ABB RobotStudio station: robotic-ABB-Cake-Simulation-Final.rspag

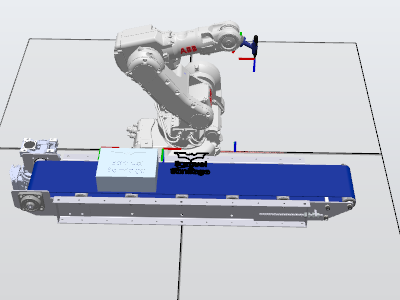
--- station ---
Station robotic-ABB-Cake (saved by RobotStudio 25.3.11371.0)
Controller IRB140_6_81
  mechanical unit ROB_1: IRB140_6_81_C_03, 6 joints, base frame (0, 0, 0) mm
Layout (positions relative to the parent item):
  - IRB140_6_81_C_03 [mechanism, from %ABB.RobotStudio.Models.IRB140%\IRB140_6_81_C_G_03.rslib] at (0, 0, 0) mm; joint values [0, -0.726, 0.4848, 0, 0.7648, 0] (rad or m)
  - Marker [mechanism] at (256.29, 0, 679.5) mm, rotated rx 180 ry 60 rz 180 deg
      TCP Marker at (50.06, 0, 105.48) mm, rotated rx 0 ry 60 rz 0 deg
      links: Marker-Tool
  - Box_Names [part] at (-315, -770, 485) mm, size 230 x 165 x 83 mm
  - Conveyor [part] at (358.05, -804.87, 88.69) mm, rotated rx 0 ry 0 rz 90 deg, size 367.7 x 1444.4 x 354.2 mm
  - SmartComponent_1 [smart component]
      signals: DI DI01, DI DI02, DI DI03, DI Conveyor_FWD, DI Conveyor_INV, DO DI_01, DO DI_02, DO DI_03
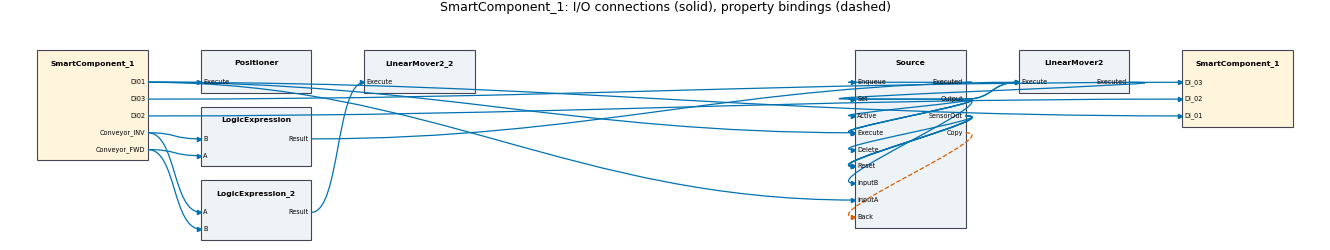
      connections:
        Source.Executed -> Queue.Enqueue
        LinearMover2.Executed -> LogicSRLatch.Set
        LogicSRLatch.Output -> Timer.Active
        Timer.Output -> LogicSRLatch_2.Set
        LogicSRLatch_2.Output -> LinearMover.Execute
        LineSensor.SensorOut -> Queue.Delete
        LineSensor.SensorOut -> Timer.Reset
        LineSensor.SensorOut -> LogicSRLatch.Reset
        LineSensor.SensorOut -> LogicSRLatch_2.Reset
        Repeater.Output -> LinearMover2.Execute
        Repeater.Output -> Source.Execute
        Timer_2.Output -> LogicGate.InputB
        LogicSRLatch_3.Output -> Source.Execute
        LogicSRLatch_3.Output -> LinearMover2.Execute
        LogicGate.Output -> LogicSRLatch_3.Set
        LineSensor.SensorOut -> LogicSRLatch_3.Reset
        SmartComponent_1.DI01 -> ?.Execute
        SmartComponent_1.DI01 -> LogicGate.InputA
        SmartComponent_1.DI03 -> SmartComponent_1.DI_03
        SmartComponent_1.DI02 -> SmartComponent_1.DI_02
        SmartComponent_1.DI01 -> SmartComponent_1.DI_01
        SmartComponent_1.Conveyor_INV -> LogicExpression.B
        SmartComponent_1.Conveyor_FWD -> LogicExpression.A
        LogicExpression.Result -> LinearMover2.Execute
        SmartComponent_1.Conveyor_INV -> LogicExpression_2.A
        SmartComponent_1.Conveyor_FWD -> LogicExpression_2.B
        LogicExpression_2.Result -> LinearMover2_2.Execute
        SmartComponent_1.DI01 -> Positioner.Execute
        Source.Copy => Queue.Back
    - LinearMover2 [smart component, from Components\LinearMover2.rslib]
        properties: Object=Box_Names; Direction=[1 0 0]; Distance=0.25; Duration=3; Reference=Global; ReferenceObject=(none)
    - LogicExpression [smart component, from Components\LogicExpression.rslib]
        properties: Expression=A AND NOT B
    - Positioner [smart component, from Components\Positioner.rslib]
        properties: Object=Box_Names; Position=[-0.315 -0.77 0.485]; Orientation=[0 0 0]; Reference=Global; ReferenceObject=(none)
    - LinearMover2_2 [smart component, from Components\LinearMover2.rslib]
        properties: Object=Box_Names; Direction=[-1 0 0]; Distance=0.5; Duration=8.5; Reference=Global; ReferenceObject=(none)
    - LogicExpression_2 [smart component, from Components\LogicExpression.rslib]
        properties: Expression=A AND NOT B
Attachment: Marker is attached to IRB140_6_81_C_03 / Link6
Attachment: Cake is attached to Box_Names
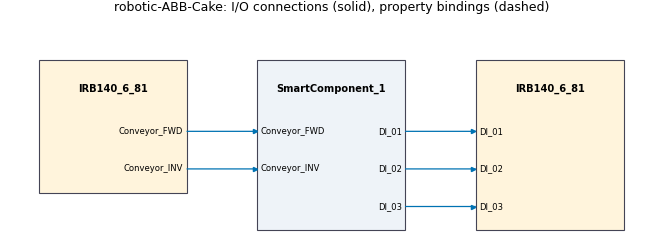
Station logic (signal -> signal, property => property):
  IRB140_6_81.Conveyor_FWD -> SmartComponent_1.Conveyor_FWD
  IRB140_6_81.Conveyor_INV -> SmartComponent_1.Conveyor_INV
  SmartComponent_1.DI_01 -> IRB140_6_81.DI_01
  SmartComponent_1.DI_02 -> IRB140_6_81.DI_02
  SmartComponent_1.DI_03 -> IRB140_6_81.DI_03

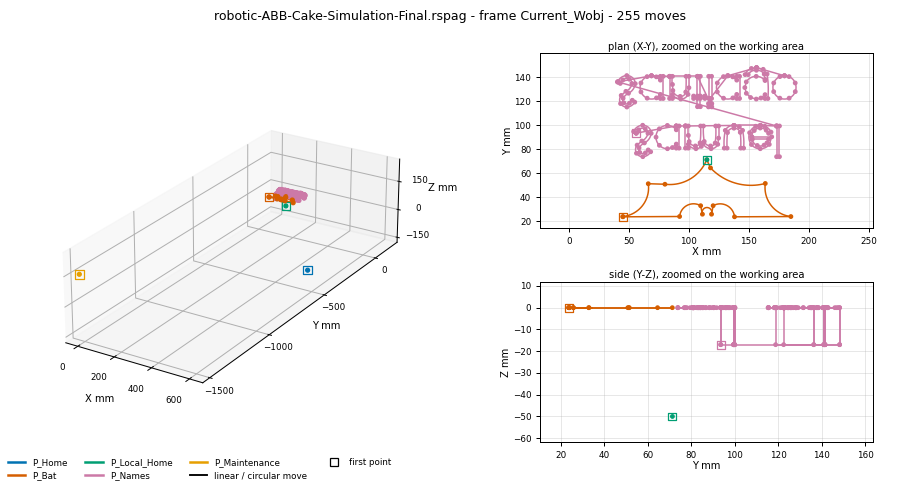
[picture p0: tool path of robotic-ABB-Cake-Simulation-Final.rspag in frame Current_Wobj, 255 of 255 moves have a stored position in this frame; points joined in program order, loops and branches not executed]
--- Controller Data/IRB140_6_81/RAPID/TASK1/PROGMOD/CalibData.mod ---
MODULE CalibData
ENDMODULE

--- Controller Data/IRB140_6_81/RAPID/TASK1/PROGMOD/Module1.mod ---
MODULE Module1
    !DATA
    !Homes
    CONST robtarget T_Home:=[[637.610974939,-605,-15.40043816],[0,0,0,1],[0,0,0,0],[9E+09,9E+09,9E+09,9E+09,9E+09,9E+09]];
    CONST robtarget T_Local_Home:=[[115.079,71.263,-50],[0.707106781,0.000000005,-0.000000005,-0.707106781],[0,0,0,0],[9E+09,9E+09,9E+09,9E+09,9E+09,9E+09]];

    !Batman Icon
    CONST robtarget Target_290:=[[44.887375283,23.575,0],[0.707106781,0,0,-0.707106781],[0,0,0,0],[9E+09,9E+09,9E+09,9E+09,9E+09,9E+09]];
    CONST robtarget Target_300:=[[92.217626762,23.834877014,0],[0.5,0,0,-0.866025404],[-1,0,-1,0],[9E+09,9E+09,9E+09,9E+09,9E+09,9E+09]];
    CONST robtarget Target_400:=[[168.340891695,33.478608179,0],[0.5,0,0,-0.866025404],[-1,0,-1,0],[9E+09,9E+09,9E+09,9E+09,9E+09,9E+09]];
    CONST robtarget Target_430:=[[118.021503486,64.425747652,0],[0.5,0,0,-0.866025404],[0,0,0,0],[9E+09,9E+09,9E+09,9E+09,9E+09,9E+09]];
    CONST robtarget Target_310:=[[97.860623741,32.777873993,0],[0.5,0,0,-0.866025404],[-1,0,-1,0],[9E+09,9E+09,9E+09,9E+09,9E+09,9E+09]];
    CONST robtarget Target_480:=[[61.659109682,33.478608179,0],[0.5,0,0,-0.866025404],[-1,0,-1,0],[9E+09,9E+09,9E+09,9E+09,9E+09,9E+09]];
    CONST robtarget Target_420:=[[135.262514114,52.897562122,0],[0.5,0,0,-0.866025404],[-1,0,-1,0],[9E+09,9E+09,9E+09,9E+09,9E+09,9E+09]];
    CONST robtarget Target_460:=[[79.985840188,50.770867258,0],[0.5,0,0,-0.866025404],[0,0,0,0],[9E+09,9E+09,9E+09,9E+09,9E+09,9E+09]];
    CONST robtarget Target_330:=[[111.283377266,25.744747734,0],[0.5,0,0,-0.866025404],[-1,0,-1,0],[9E+09,9E+09,9E+09,9E+09,9E+09,9E+09]];
    CONST robtarget Target_380:=[[138.079373741,23.575,0],[0.5,0,0,-0.866025404],[0,0,0,0],[9E+09,9E+09,9E+09,9E+09,9E+09,9E+09]];
    CONST robtarget Target_340:=[[112.525,30.426625252,0],[0.5,0,0,-0.866025404],[-1,0,-1,0],[9E+09,9E+09,9E+09,9E+09,9E+09,9E+09]];
    CONST robtarget Target_490:=[[44.854375315,23.789501762,0],[0.707106781,0,0,-0.707106781],[0,0,0,0],[9E+09,9E+09,9E+09,9E+09,9E+09,9E+09]];
    CONST robtarget Target_360:=[[120.205747986,32.852127266,0],[0.5,0,0,-0.866025404],[-1,0,-1,0],[9E+09,9E+09,9E+09,9E+09,9E+09,9E+09]];
    CONST robtarget Target_350:=[[118.898123741,25.740625,0],[0.5,0,0,-0.866025404],[0,0,0,0],[9E+09,9E+09,9E+09,9E+09,9E+09,9E+09]];
    CONST robtarget Target_370:=[[132.139376259,32.777873993,0],[0.5,0,0,-0.866025404],[-1,0,-1,0],[9E+09,9E+09,9E+09,9E+09,9E+09,9E+09]];
    CONST robtarget Target_410:=[[163.773995972,51.414627266,0],[0.5,0,0,-0.866025404],[0,0,0,0],[9E+09,9E+09,9E+09,9E+09,9E+09,9E+09]];
    CONST robtarget Target_470:=[[66.061000252,51.208377266,0],[0.5,0,0,-0.866025404],[-1,0,-1,0],[9E+09,9E+09,9E+09,9E+09,9E+09,9E+09]];
    CONST robtarget Target_320:=[[109.794252014,32.852127266,0],[0.5,0,0,-0.866025404],[0,0,0,0],[9E+09,9E+09,9E+09,9E+09,9E+09,9E+09]];
    CONST robtarget Target_440:=[[114.884500504,71.210504532,0],[0.5,0,0,-0.866025404],[-1,0,-1,0],[9E+09,9E+09,9E+09,9E+09,9E+09,9E+09]];
    CONST robtarget Target_450:=[[101.522546531,55.448907324,0],[0.5,0,0,-0.866025404],[-1,0,-1,0],[9E+09,9E+09,9E+09,9E+09,9E+09,9E+09]];
    CONST robtarget Target_390:=[[185.145619965,23.789501762,0],[0.5,0,0,-0.866025404],[-1,0,-1,0],[9E+09,9E+09,9E+09,9E+09,9E+09,9E+09]];

    !Nombres
    CONST robtarget Names_00:=[[55.976,93.47,-17],[0.707106781,0,0,-0.707106781],[0,0,0,0],[9E+09,9E+09,9E+09,9E+09,9E+09,9E+09]];
    CONST robtarget Names_10:=[[55.976,93.47,0],[0.707106781,0,0,-0.707106781],[-1,-1,0,0],[9E+09,9E+09,9E+09,9E+09,9E+09,9E+09]];
    CONST robtarget Names_20:=[[53.851,94.745,0],[0.707106781,0,0,-0.707106781],[-1,-1,0,0],[9E+09,9E+09,9E+09,9E+09,9E+09,9E+09]];
    CONST robtarget Names_30:=[[57.267,98.815,0],[0.707106781,0,0,-0.707106781],[-1,-1,0,0],[9E+09,9E+09,9E+09,9E+09,9E+09,9E+09]];
    CONST robtarget Names_40:=[[61.397,100.031,0],[0.707106781,0,0,-0.707106781],[-1,-1,0,0],[9E+09,9E+09,9E+09,9E+09,9E+09,9E+09]];
    CONST robtarget Names_50:=[[66.419,98.025,0],[0.707106781,0,0,-0.707106781],[-1,-1,0,0],[9E+09,9E+09,9E+09,9E+09,9E+09,9E+09]];
    CONST robtarget Names_60:=[[68.484,93.3,0],[0.707106781,0,0,-0.707106781],[-1,-1,0,0],[9E+09,9E+09,9E+09,9E+09,9E+09,9E+09]];
    CONST robtarget Names_70:=[[67.277,89.545,0],[0.707106781,0,0,-0.707106781],[-1,-1,0,0],[9E+09,9E+09,9E+09,9E+09,9E+09,9E+09]];
    CONST robtarget Names_80:=[[62.825,85.279,0],[0.707106781,0,0,-0.707106781],[-1,-1,0,0],[9E+09,9E+09,9E+09,9E+09,9E+09,9E+09]];
    CONST robtarget Names_90:=[[59.596,82.78,0],[0.707106781,0,0,-0.707106781],[-1,-1,0,0],[9E+09,9E+09,9E+09,9E+09,9E+09,9E+09]];
    CONST robtarget Names_100:=[[58.355,81.115,0],[0.707106781,0,0,-0.707106781],[-1,-1,0,0],[9E+09,9E+09,9E+09,9E+09,9E+09,9E+09]];
    CONST robtarget Names_110:=[[58.015,79.534,0],[0.707106781,0,0,-0.707106781],[-1,-1,0,0],[9E+09,9E+09,9E+09,9E+09,9E+09,9E+09]];
    CONST robtarget Names_120:=[[58.975,77.274,0],[0.707106781,0,0,-0.707106781],[-1,-1,0,0],[9E+09,9E+09,9E+09,9E+09,9E+09,9E+09]];
    CONST robtarget Names_130:=[[61.448,76.356,0],[0.707106781,0,0,-0.707106781],[-1,-1,0,0],[9E+09,9E+09,9E+09,9E+09,9E+09,9E+09]];
    CONST robtarget Names_140:=[[63.615,76.951,0],[0.707106781,0,0,-0.707106781],[-1,-1,0,0],[9E+09,9E+09,9E+09,9E+09,9E+09,9E+09]];
    CONST robtarget Names_150:=[[66.02,79.415,0],[0.707106781,0,0,-0.707106781],[-1,-1,0,0],[9E+09,9E+09,9E+09,9E+09,9E+09,9E+09]];
    CONST robtarget Names_160:=[[68.059,77.869,0],[0.707106781,0,0,-0.707106781],[-1,-1,0,0],[9E+09,9E+09,9E+09,9E+09,9E+09,9E+09]];
    CONST robtarget Names_170:=[[64.805,74.648,0],[0.707106781,0,0,-0.707106781],[-1,-1,0,0],[9E+09,9E+09,9E+09,9E+09,9E+09,9E+09]];
    CONST robtarget Names_180:=[[61.499,73.773,0],[0.707106781,0,0,-0.707106781],[-1,-1,0,0],[9E+09,9E+09,9E+09,9E+09,9E+09,9E+09]];
    CONST robtarget Names_190:=[[58.414,74.546,0],[0.707106781,0,0,-0.707106781],[-1,-1,0,0],[9E+09,9E+09,9E+09,9E+09,9E+09,9E+09]];
    CONST robtarget Names_200:=[[56.213,76.662,0],[0.707106781,0,0,-0.707106781],[-1,-1,0,0],[9E+09,9E+09,9E+09,9E+09,9E+09,9E+09]];
    CONST robtarget Names_210:=[[55.432,79.636,0],[0.707106781,0,0,-0.707106781],[-1,-1,0,0],[9E+09,9E+09,9E+09,9E+09,9E+09,9E+09]];
    CONST robtarget Names_220:=[[56.757,83.46,0],[0.707106781,0,0,-0.707106781],[-1,-1,0,0],[9E+09,9E+09,9E+09,9E+09,9E+09,9E+09]];
    CONST robtarget Names_230:=[[60.649,86.876,0],[0.707106781,0,0,-0.707106781],[-1,-1,0,0],[9E+09,9E+09,9E+09,9E+09,9E+09,9E+09]];
    CONST robtarget Names_240:=[[64.932,90.887,0],[0.707106781,0,0,-0.707106781],[-1,-1,0,0],[9E+09,9E+09,9E+09,9E+09,9E+09,9E+09]];
    CONST robtarget Names_250:=[[65.782,93.351,0],[0.707106781,0,0,-0.707106781],[-1,-1,0,0],[9E+09,9E+09,9E+09,9E+09,9E+09,9E+09]];
    CONST robtarget Names_260:=[[65.204,95.442,0],[0.707106781,0,0,-0.707106781],[-1,-1,0,0],[9E+09,9E+09,9E+09,9E+09,9E+09,9E+09]];
    CONST robtarget Names_270:=[[63.521,97.014,0],[0.707106781,0,0,-0.707106781],[-1,-1,0,0],[9E+09,9E+09,9E+09,9E+09,9E+09,9E+09]];
    CONST robtarget Names_280:=[[61.159,97.6,0],[0.707106781,0,0,-0.707106781],[-1,-1,0,0],[9E+09,9E+09,9E+09,9E+09,9E+09,9E+09]];
    CONST robtarget Names_290:=[[58.019,96.283,0],[0.707106781,0,0,-0.707106781],[-1,-1,0,0],[9E+09,9E+09,9E+09,9E+09,9E+09,9E+09]];
    CONST robtarget Names_300:=[[55.976,93.47,0],[0.707106781,0,0,-0.707106781],[-1,-1,0,0],[9E+09,9E+09,9E+09,9E+09,9E+09,9E+09]];
    CONST robtarget Names_310:=[[55.976,93.47,-17],[0.707106781,0,0,-0.707106781],[-1,-1,0,0],[9E+09,9E+09,9E+09,9E+09,9E+09,9E+09]];
    CONST robtarget Names_320:=[[89.456,99.402,-17],[0.608761429,0,0,-0.79335334],[-1,0,-1,0],[9E+09,9E+09,9E+09,9E+09,9E+09,9E+09]];
    CONST robtarget Names_330:=[[89.456,99.402,0],[0.608761429,0,0,-0.79335334],[-1,0,-1,0],[9E+09,9E+09,9E+09,9E+09,9E+09,9E+09]];
    CONST robtarget Names_340:=[[89.456,96.224,0],[0.608761429,0,0,-0.79335334],[-1,0,-1,0],[9E+09,9E+09,9E+09,9E+09,9E+09,9E+09]];
    CONST robtarget Names_350:=[[86.1,98.96,0],[0.608761429,0,0,-0.79335334],[-1,0,-1,0],[9E+09,9E+09,9E+09,9E+09,9E+09,9E+09]];
    CONST robtarget Names_360:=[[82.029,99.878,0],[0.608761429,0,0,-0.79335334],[-1,0,-1,0],[9E+09,9E+09,9E+09,9E+09,9E+09,9E+09]];
    CONST robtarget Names_370:=[[78.378,99.161,0],[0.608761429,0,0,-0.79335334],[-1,0,-1,0],[9E+09,9E+09,9E+09,9E+09,9E+09,9E+09]];
    CONST robtarget Names_380:=[[75.325,97.031,0],[0.608761429,0,0,-0.79335334],[-1,0,-1,0],[9E+09,9E+09,9E+09,9E+09,9E+09,9E+09]];
    CONST robtarget Names_390:=[[73.231,93.852,0],[0.608761429,0,0,-0.79335334],[-1,0,-1,0],[9E+09,9E+09,9E+09,9E+09,9E+09,9E+09]];
    CONST robtarget Names_400:=[[72.546,90.105,0],[0.608761429,0,0,-0.79335334],[-1,0,-1,0],[9E+09,9E+09,9E+09,9E+09,9E+09,9E+09]];
    CONST robtarget Names_410:=[[73.247,86.401,0],[0.608761429,0,0,-0.79335334],[-1,0,-1,0],[9E+09,9E+09,9E+09,9E+09,9E+09,9E+09]];
    CONST robtarget Names_420:=[[75.35,83.273,0],[0.608761429,0,0,-0.79335334],[-1,0,-1,0],[9E+09,9E+09,9E+09,9E+09,9E+09,9E+09]];
    CONST robtarget Names_430:=[[78.428,81.149,0],[0.608761429,0,0,-0.79335334],[-1,0,-1,0],[9E+09,9E+09,9E+09,9E+09,9E+09,9E+09]];
    CONST robtarget Names_440:=[[82.097,80.435,0],[0.608761429,0,0,-0.79335334],[-1,0,-1,0],[9E+09,9E+09,9E+09,9E+09,9E+09,9E+09]];
    CONST robtarget Names_450:=[[86.219,81.404,0],[0.608761429,0,0,-0.79335334],[-1,0,-1,0],[9E+09,9E+09,9E+09,9E+09,9E+09,9E+09]];
    CONST robtarget Names_460:=[[89.456,84.31,0],[0.608761429,0,0,-0.79335334],[-1,0,-1,0],[9E+09,9E+09,9E+09,9E+09,9E+09,9E+09]];
    CONST robtarget Names_470:=[[89.456,80.911,0],[0.608761429,0,0,-0.79335334],[-1,0,-1,0],[9E+09,9E+09,9E+09,9E+09,9E+09,9E+09]];
    CONST robtarget Names_480:=[[91.801,80.911,0],[0.608761429,0,0,-0.79335334],[-1,0,-1,0],[9E+09,9E+09,9E+09,9E+09,9E+09,9E+09]];
    CONST robtarget Names_490:=[[91.801,99.402,0],[0.608761429,0,0,-0.79335334],[-1,0,-1,0],[9E+09,9E+09,9E+09,9E+09,9E+09,9E+09]];
    CONST robtarget Names_500:=[[89.456,99.402,0],[0.608761429,0,0,-0.79335334],[-1,0,-1,0],[9E+09,9E+09,9E+09,9E+09,9E+09,9E+09]];
    CONST robtarget Names_510:=[[89.456,99.402,-17],[0.608761429,0,0,-0.79335334],[-1,0,-1,0],[9E+09,9E+09,9E+09,9E+09,9E+09,9E+09]];
    CONST robtarget Names_520:=[[97.138,99.402,-17],[0.608761429,0,0,-0.79335334],[-1,0,-1,0],[9E+09,9E+09,9E+09,9E+09,9E+09,9E+09]];
    CONST robtarget Names_530:=[[97.138,99.402,0],[0.608761429,0,0,-0.79335334],[-1,0,-1,0],[9E+09,9E+09,9E+09,9E+09,9E+09,9E+09]];
    CONST robtarget Names_540:=[[97.138,80.911,0],[0.608761429,0,0,-0.79335334],[-1,0,-1,0],[9E+09,9E+09,9E+09,9E+09,9E+09,9E+09]];
    CONST robtarget Names_550:=[[99.517,80.911,0],[0.608761429,0,0,-0.79335334],[-1,0,-1,0],[9E+09,9E+09,9E+09,9E+09,9E+09,9E+09]];
    CONST robtarget Names_560:=[[99.517,84.106,0],[0.608761429,0,0,-0.79335334],[-1,0,-1,0],[9E+09,9E+09,9E+09,9E+09,9E+09,9E+09]];
    CONST robtarget Names_570:=[[102.07,81.523,0],[0.608761429,0,0,-0.79335334],[-1,0,-1,0],[9E+09,9E+09,9E+09,9E+09,9E+09,9E+09]];
    CONST robtarget Names_580:=[[105.864,80.435,0],[0.608761429,0,0,-0.79335334],[-1,0,-1,0],[9E+09,9E+09,9E+09,9E+09,9E+09,9E+09]];
    CONST robtarget Names_590:=[[108.416,80.962,0],[0.608761429,0,0,-0.79335334],[-1,0,-1,0],[9E+09,9E+09,9E+09,9E+09,9E+09,9E+09]];
    CONST robtarget Names_600:=[[110.39,82.364,0],[0.608761429,0,0,-0.79335334],[-1,0,-1,0],[9E+09,9E+09,9E+09,9E+09,9E+09,9E+09]];
    CONST robtarget Names_610:=[[111.717,84.871,0],[0.608761429,0,0,-0.79335334],[-1,0,-1,0],[9E+09,9E+09,9E+09,9E+09,9E+09,9E+09]];
    CONST robtarget Names_620:=[[114.684,81.565,0],[0.608761429,0,0,-0.79335334],[-1,0,-1,0],[9E+09,9E+09,9E+09,9E+09,9E+09,9E+09]];
    CONST robtarget Names_630:=[[118.516,80.435,0],[0.608761429,0,0,-0.79335334],[-1,0,-1,0],[9E+09,9E+09,9E+09,9E+09,9E+09,9E+09]];
    CONST robtarget Names_640:=[[121.898,81.404,0],[0.608761429,0,0,-0.79335334],[-1,0,-1,0],[9E+09,9E+09,9E+09,9E+09,9E+09,9E+09]];
    CONST robtarget Names_650:=[[124.077,84.106,0],[0.608761429,0,0,-0.79335334],[-1,0,-1,0],[9E+09,9E+09,9E+09,9E+09,9E+09,9E+09]];
    CONST robtarget Names_660:=[[124.789,89.307,0],[0.608761429,0,0,-0.79335334],[-1,0,-1,0],[9E+09,9E+09,9E+09,9E+09,9E+09,9E+09]];
    CONST robtarget Names_670:=[[124.789,99.402,0],[0.608761429,0,0,-0.79335334],[-1,0,-1,0],[9E+09,9E+09,9E+09,9E+09,9E+09,9E+09]];
    CONST robtarget Names_680:=[[122.359,99.402,0],[0.608761429,0,0,-0.79335334],[-1,0,-1,0],[9E+09,9E+09,9E+09,9E+09,9E+09,9E+09]];
    CONST robtarget Names_690:=[[122.359,89.307,0],[0.608761429,0,0,-0.79335334],[-1,0,-1,0],[9E+09,9E+09,9E+09,9E+09,9E+09,9E+09]];
    CONST robtarget Names_700:=[[121.936,85.219,0],[0.608761429,0,0,-0.79335334],[-1,0,-1,0],[9E+09,9E+09,9E+09,9E+09,9E+09,9E+09]];
    CONST robtarget Names_710:=[[120.487,83.426,0],[0.608761429,0,0,-0.79335334],[-1,0,-1,0],[9E+09,9E+09,9E+09,9E+09,9E+09,9E+09]];
    CONST robtarget Names_720:=[[118.039,82.746,0],[0.608761429,0,0,-0.79335334],[-1,0,-1,0],[9E+09,9E+09,9E+09,9E+09,9E+09,9E+09]];
    CONST robtarget Names_730:=[[114.88,83.766,0],[0.608761429,0,0,-0.79335334],[-1,0,-1,0],[9E+09,9E+09,9E+09,9E+09,9E+09,9E+09]];
    CONST robtarget Names_740:=[[112.788,86.485,0],[0.608761429,0,0,-0.79335334],[-1,0,-1,0],[9E+09,9E+09,9E+09,9E+09,9E+09,9E+09]];
    CONST robtarget Names_750:=[[112.128,92.162,0],[0.608761429,0,0,-0.79335334],[-1,0,-1,0],[9E+09,9E+09,9E+09,9E+09,9E+09,9E+09]];
    CONST robtarget Names_760:=[[112.128,99.402,0],[0.608761429,0,0,-0.79335334],[-1,0,-1,0],[9E+09,9E+09,9E+09,9E+09,9E+09,9E+09]];
    CONST robtarget Names_770:=[[109.748,99.402,0],[0.608761429,0,0,-0.79335334],[-1,0,-1,0],[9E+09,9E+09,9E+09,9E+09,9E+09,9E+09]];
    CONST robtarget Names_780:=[[109.748,89.935,0],[0.608761429,0,0,-0.79335334],[-1,0,-1,0],[9E+09,9E+09,9E+09,9E+09,9E+09,9E+09]];
    CONST robtarget Names_790:=[[109.332,85.389,0],[0.608761429,0,0,-0.79335334],[-1,0,-1,0],[9E+09,9E+09,9E+09,9E+09,9E+09,9E+09]];
    CONST robtarget Names_800:=[[107.879,83.469,0],[0.608761429,0,0,-0.79335334],[-1,0,-1,0],[9E+09,9E+09,9E+09,9E+09,9E+09,9E+09]];
    CONST robtarget Names_810:=[[105.415,82.746,0],[0.608761429,0,0,-0.79335334],[-1,0,-1,0],[9E+09,9E+09,9E+09,9E+09,9E+09,9E+09]];
    CONST robtarget Names_820:=[[102.33,83.741,0],[0.608761429,0,0,-0.79335334],[-1,0,-1,0],[9E+09,9E+09,9E+09,9E+09,9E+09,9E+09]];
    CONST robtarget Names_830:=[[100.206,86.417,0],[0.608761429,0,0,-0.79335334],[-1,0,-1,0],[9E+09,9E+09,9E+09,9E+09,9E+09,9E+09]];
    CONST robtarget Names_840:=[[99.517,91.567,0],[0.608761429,0,0,-0.79335334],[-1,0,-1,0],[9E+09,9E+09,9E+09,9E+09,9E+09,9E+09]];
    CONST robtarget Names_850:=[[99.517,99.402,0],[0.608761429,0,0,-0.79335334],[-1,0,-1,0],[9E+09,9E+09,9E+09,9E+09,9E+09,9E+09]];
    CONST robtarget Names_860:=[[97.138,99.402,0],[0.608761429,0,0,-0.79335334],[-1,0,-1,0],[9E+09,9E+09,9E+09,9E+09,9E+09,9E+09]];
    CONST robtarget Names_870:=[[97.138,99.402,-17],[0.608761429,0,0,-0.79335334],[-1,0,-1,0],[9E+09,9E+09,9E+09,9E+09,9E+09,9E+09]];
    CONST robtarget Names_880:=[[137.604,99.878,-17],[0.5,0,0,-0.866025404],[-1,0,-1,0],[9E+09,9E+09,9E+09,9E+09,9E+09,9E+09]];
    CONST robtarget Names_890:=[[137.604,99.878,0],[0.5,0,0,-0.866025404],[-1,0,-1,0],[9E+09,9E+09,9E+09,9E+09,9E+09,9E+09]];
    CONST robtarget Names_900:=[[133.091,98.781,0],[0.5,0,0,-0.866025404],[-1,0,-1,0],[9E+09,9E+09,9E+09,9E+09,9E+09,9E+09]];
    CONST robtarget Names_910:=[[130.389,95.722,0],[0.5,0,0,-0.866025404],[-1,0,-1,0],[9E+09,9E+09,9E+09,9E+09,9E+09,9E+09]];
    CONST robtarget Names_920:=[[129.497,89.816,0],[0.5,0,0,-0.866025404],[-1,0,-1,0],[9E+09,9E+09,9E+09,9E+09,9E+09,9E+09]];
    CONST robtarget Names_930:=[[129.497,80.911,0],[0.5,0,0,-0.866025404],[-1,0,-1,0],[9E+09,9E+09,9E+09,9E+09,9E+09,9E+09]];
    CONST robtarget Names_940:=[[131.876,80.911,0],[0.5,0,0,-0.866025404],[-1,0,-1,0],[9E+09,9E+09,9E+09,9E+09,9E+09,9E+09]];
    CONST robtarget Names_950:=[[131.876,89.545,0],[0.5,0,0,-0.866025404],[-1,0,-1,0],[9E+09,9E+09,9E+09,9E+09,9E+09,9E+09]];
    CONST robtarget Names_960:=[[132.217,93.895,0],[0.5,0,0,-0.866025404],[-1,0,-1,0],[9E+09,9E+09,9E+09,9E+09,9E+09,9E+09]];
    CONST robtarget Names_970:=[[134.166,96.581,0],[0.5,0,0,-0.866025404],[-1,0,-1,0],[9E+09,9E+09,9E+09,9E+09,9E+09,9E+09]];
    CONST robtarget Names_980:=[[137.595,97.566,0],[0.5,0,0,-0.866025404],[-1,0,-1,0],[9E+09,9E+09,9E+09,9E+09,9E+09,9E+09]];
    CONST robtarget Names_990:=[[140.974,96.606,0],[0.5,0,0,-0.866025404],[-1,0,-1,0],[9E+09,9E+09,9E+09,9E+09,9E+09,9E+09]];
    CONST robtarget Names_1000:=[[142.889,94.082,0],[0.5,0,0,-0.866025404],[-1,0,-1,0],[9E+09,9E+09,9E+09,9E+09,9E+09,9E+09]];
    CONST robtarget Names_1010:=[[143.246,89.545,0],[0.5,0,0,-0.866025404],[-1,0,-1,0],[9E+09,9E+09,9E+09,9E+09,9E+09,9E+09]];
    CONST robtarget Names_1020:=[[143.246,80.911,0],[0.5,0,0,-0.866025404],[-1,0,-1,0],[9E+09,9E+09,9E+09,9E+09,9E+09,9E+09]];
    CONST robtarget Names_1030:=[[145.676,80.911,0],[0.5,0,0,-0.866025404],[-1,0,-1,0],[9E+09,9E+09,9E+09,9E+09,9E+09,9E+09]];
    CONST robtarget Names_1040:=[[145.676,89.986,0],[0.5,0,0,-0.866025404],[-1,0,-1,0],[9E+09,9E+09,9E+09,9E+09,9E+09,9E+09]];
    CONST robtarget Names_1050:=[[144.784,95.748,0],[0.5,0,0,-0.866025404],[-1,0,-1,0],[9E+09,9E+09,9E+09,9E+09,9E+09,9E+09]];
    CONST robtarget Names_1060:=[[142.099,98.781,0],[0.5,0,0,-0.866025404],[-1,0,-1,0],[9E+09,9E+09,9E+09,9E+09,9E+09,9E+09]];
    CONST robtarget Names_1070:=[[137.604,99.878,0],[0.5,0,0,-0.866025404],[-1,0,-1,0],[9E+09,9E+09,9E+09,9E+09,9E+09,9E+09]];
    CONST robtarget Names_1080:=[[137.604,99.878,-17],[0.5,0,0,-0.866025404],[-1,0,-1,0],[9E+09,9E+09,9E+09,9E+09,9E+09,9E+09]];
    CONST robtarget Names_1090:=[[159.689,99.878,-17],[0.5,0,0,-0.866025404],[-1,0,-1,0],[9E+09,9E+09,9E+09,9E+09,9E+09,9E+09]];
    CONST robtarget Names_1100:=[[159.689,99.878,0],[0.5,0,0,-0.866025404],[-1,0,-1,0],[9E+09,9E+09,9E+09,9E+09,9E+09,9E+09]];
    CONST robtarget Names_1110:=[[155.805,99.199,0],[0.5,0,0,-0.866025404],[-1,0,-1,0],[9E+09,9E+09,9E+09,9E+09,9E+09,9E+09]];
    CONST robtarget Names_1120:=[[152.613,96.912,0],[0.5,0,0,-0.866025404],[-1,0,-1,0],[9E+09,9E+09,9E+09,9E+09,9E+09,9E+09]];
    CONST robtarget Names_1130:=[[150.715,93.795,0],[0.5,0,0,-0.866025404],[-1,0,-1,0],[9E+09,9E+09,9E+09,9E+09,9E+09,9E+09]];
    CONST robtarget Names_1140:=[[150.061,90.207,0],[0.5,0,0,-0.866025404],[-1,0,-1,0],[9E+09,9E+09,9E+09,9E+09,9E+09,9E+09]];
    CONST robtarget Names_1150:=[[152.221,83.936,0],[0.5,0,0,-0.866025404],[-1,0,-1,0],[9E+09,9E+09,9E+09,9E+09,9E+09,9E+09]];
    CONST robtarget Names_1160:=[[155.459,81.294,0],[0.5,0,0,-0.866025404],[-1,0,-1,0],[9E+09,9E+09,9E+09,9E+09,9E+09,9E+09]];
    CONST robtarget Names_1170:=[[159.553,80.435,0],[0.5,0,0,-0.866025404],[-1,0,-1,0],[9E+09,9E+09,9E+09,9E+09,9E+09,9E+09]];
    CONST robtarget Names_1180:=[[163.767,81.313,0],[0.5,0,0,-0.866025404],[-1,0,-1,0],[9E+09,9E+09,9E+09,9E+09,9E+09,9E+09]];
    CONST robtarget Names_1190:=[[167.106,84.021,0],[0.5,0,0,-0.866025404],[-1,0,-1,0],[9E+09,9E+09,9E+09,9E+09,9E+09,9E+09]];
    CONST robtarget Names_1200:=[[169.147,90.343,0],[0.5,0,0,-0.866025404],[-1,0,-1,0],[9E+09,9E+09,9E+09,9E+09,9E+09,9E+09]];
    CONST robtarget Names_1210:=[[152.508,90.343,0],[0.5,0,0,-0.866025404],[-1,0,-1,0],[9E+09,9E+09,9E+09,9E+09,9E+09,9E+09]];
    CONST robtarget Names_1220:=[[152.746,88.287,0],[0.5,0,0,-0.866025404],[-1,0,-1,0],[9E+09,9E+09,9E+09,9E+09,9E+09,9E+09]];
    CONST robtarget Names_1230:=[[154.907,84.463,0],[0.5,0,0,-0.866025404],[-1,0,-1,0],[9E+09,9E+09,9E+09,9E+09,9E+09,9E+09]];
    CONST robtarget Names_1240:=[[157.079,83.141,0],[0.5,0,0,-0.866025404],[-1,0,-1,0],[9E+09,9E+09,9E+09,9E+09,9E+09,9E+09]];
    CONST robtarget Names_1250:=[[159.587,82.712,0],[0.5,0,0,-0.866025404],[-1,0,-1,0],[9E+09,9E+09,9E+09,9E+09,9E+09,9E+09]];
    CONST robtarget Names_1260:=[[162.735,83.409,0],[0.5,0,0,-0.866025404],[-1,0,-1,0],[9E+09,9E+09,9E+09,9E+09,9E+09,9E+09]];
    CONST robtarget Names_1270:=[[165.143,85.245,0],[0.5,0,0,-0.866025404],[-1,0,-1,0],[9E+09,9E+09,9E+09,9E+09,9E+09,9E+09]];
    CONST robtarget Names_1280:=[[166.53,88.287,0],[0.5,0,0,-0.866025404],[-1,0,-1,0],[9E+09,9E+09,9E+09,9E+09,9E+09,9E+09]];
    CONST robtarget Names_1290:=[[152.746,88.287,0],[0.5,0,0,-0.866025404],[-1,0,-1,0],[9E+09,9E+09,9E+09,9E+09,9E+09,9E+09]];
    CONST robtarget Names_1300:=[[152.508,90.343,0],[0.5,0,0,-0.866025404],[-1,0,-1,0],[9E+09,9E+09,9E+09,9E+09,9E+09,9E+09]];
    CONST robtarget Names_1310:=[[153.023,93.189,0],[0.5,0,0,-0.866025404],[-1,0,-1,0],[9E+09,9E+09,9E+09,9E+09,9E+09,9E+09]];
    CONST robtarget Names_1320:=[[154.567,95.625,0],[0.5,0,0,-0.866025404],[-1,0,-1,0],[9E+09,9E+09,9E+09,9E+09,9E+09,9E+09]];
    CONST robtarget Names_1330:=[[156.807,97.176,0],[0.5,0,0,-0.866025404],[-1,0,-1,0],[9E+09,9E+09,9E+09,9E+09,9E+09,9E+09]];
    CONST robtarget Names_1340:=[[159.485,97.685,0],[0.5,0,0,-0.866025404],[-1,0,-1,0],[9E+09,9E+09,9E+09,9E+09,9E+09,9E+09]];
    CONST robtarget Names_1350:=[[162.233,97.194,0],[0.5,0,0,-0.866025404],[-1,0,-1,0],[9E+09,9E+09,9E+09,9E+09,9E+09,9E+09]];
    CONST robtarget Names_1360:=[[164.505,95.891,0],[0.5,0,0,-0.866025404],[-1,0,-1,0],[9E+09,9E+09,9E+09,9E+09,9E+09,9E+09]];
    CONST robtarget Names_1370:=[[166.53,93.266,0],[0.5,0,0,-0.866025404],[-1,0,-1,0],[9E+09,9E+09,9E+09,9E+09,9E+09,9E+09]];
    CONST robtarget Names_1380:=[[168.535,94.32,0],[0.5,0,0,-0.866025404],[-1,0,-1,0],[9E+09,9E+09,9E+09,9E+09,9E+09,9E+09]];
    CONST robtarget Names_1390:=[[166.256,97.447,0],[0.5,0,0,-0.866025404],[-1,0,-1,0],[9E+09,9E+09,9E+09,9E+09,9E+09,9E+09]];
    CONST robtarget Names_1400:=[[163.347,99.257,0],[0.5,0,0,-0.866025404],[-1,0,-1,0],[9E+09,9E+09,9E+09,9E+09,9E+09,9E+09]];
    CONST robtarget Names_1410:=[[159.689,99.878,0],[0.5,0,0,-0.866025404],[-1,0,-1,0],[9E+09,9E+09,9E+09,9E+09,9E+09,9E+09]];
    CONST robtarget Names_1420:=[[159.689,99.878,-17],[0.5,0,0,-0.866025404],[-1,0,-1,0],[9E+09,9E+09,9E+09,9E+09,9E+09,9E+09]];
    CONST robtarget Names_1430:=[[173.226,99.402,-17],[0.382683432,0,0,-0.923879533],[-1,0,-1,0],[9E+09,9E+09,9E+09,9E+09,9E+09,9E+09]];
    CONST robtarget Names_1440:=[[173.226,99.402,0],[0.382683432,0,0,-0.923879533],[-1,0,-1,0],[9E+09,9E+09,9E+09,9E+09,9E+09,9E+09]];
    CONST robtarget Names_1450:=[[173.226,73.773,0],[0.382683432,0,0,-0.923879533],[-1,0,-1,0],[9E+09,9E+09,9E+09,9E+09,9E+09,9E+09]];
    CONST robtarget Names_1460:=[[175.605,73.773,0],[0.382683432,0,0,-0.923879533],[-1,0,-1,0],[9E+09,9E+09,9E+09,9E+09,9E+09,9E+09]];
    CONST robtarget Names_1470:=[[175.605,99.402,0],[0.382683432,0,0,-0.923879533],[-1,0,-1,0],[9E+09,9E+09,9E+09,9E+09,9E+09,9E+09]];
    CONST robtarget Names_1480:=[[173.226,99.402,0],[0.382683432,0,0,-0.923879533],[-1,0,-1,0],[9E+09,9E+09,9E+09,9E+09,9E+09,9E+09]];
    CONST robtarget Names_1490:=[[173.226,99.402,-17],[0.382683432,0,0,-0.923879533],[-1,0,-1,0],[9E+09,9E+09,9E+09,9E+09,9E+09,9E+09]];
    CONST robtarget Names_1500:=[[40.561,136.213,-17],[0.707106781,0,0,-0.707106781],[-1,-1,0,0],[9E+09,9E+09,9E+09,9E+09,9E+09,9E+09]];
    CONST robtarget Names_1510:=[[40.561,136.213,0],[0.707106781,0,0,-0.707106781],[-1,-1,0,0],[9E+09,9E+09,9E+09,9E+09,9E+09,9E+09]];
    CONST robtarget Names_1520:=[[43.977,140.284,0],[0.707106781,0,0,-0.707106781],[-1,-1,0,0],[9E+09,9E+09,9E+09,9E+09,9E+09,9E+09]];
    CONST robtarget Names_1530:=[[48.107,141.499,0],[0.707106781,0,0,-0.707106781],[-1,-1,0,0],[9E+09,9E+09,9E+09,9E+09,9E+09,9E+09]];
    CONST robtarget Names_1540:=[[53.129,139.494,0],[0.707106781,0,0,-0.707106781],[-1,-1,0,0],[9E+09,9E+09,9E+09,9E+09,9E+09,9E+09]];
    CONST robtarget Names_1550:=[[55.194,134.769,0],[0.707106781,0,0,-0.707106781],[-1,-1,0,0],[9E+09,9E+09,9E+09,9E+09,9E+09,9E+09]];
    CONST robtarget Names_1560:=[[53.987,131.013,0],[0.707106781,0,0,-0.707106781],[-1,-1,0,0],[9E+09,9E+09,9E+09,9E+09,9E+09,9E+09]];
    CONST robtarget Names_1570:=[[49.534,126.747,0],[0.707106781,0,0,-0.707106781],[-1,-1,0,0],[9E+09,9E+09,9E+09,9E+09,9E+09,9E+09]];
    CONST robtarget Names_1580:=[[46.305,124.249,0],[0.707106781,0,0,-0.707106781],[-1,-1,0,0],[9E+09,9E+09,9E+09,9E+09,9E+09,9E+09]];
    CONST robtarget Names_1590:=[[45.065,122.583,0],[0.707106781,0,0,-0.707106781],[-1,-1,0,0],[9E+09,9E+09,9E+09,9E+09,9E+09,9E+09]];
    CONST robtarget Names_1600:=[[44.725,121.003,0],[0.707106781,0,0,-0.707106781],[-1,-1,0,0],[9E+09,9E+09,9E+09,9E+09,9E+09,9E+09]];
    CONST robtarget Names_1610:=[[45.685,118.742,0],[0.707106781,0,0,-0.707106781],[-1,-1,0,0],[9E+09,9E+09,9E+09,9E+09,9E+09,9E+09]];
    CONST robtarget Names_1620:=[[48.158,117.825,0],[0.707106781,0,0,-0.707106781],[-1,-1,0,0],[9E+09,9E+09,9E+09,9E+09,9E+09,9E+09]];
    CONST robtarget Names_1630:=[[50.325,118.419,0],[0.707106781,0,0,-0.707106781],[-1,-1,0,0],[9E+09,9E+09,9E+09,9E+09,9E+09,9E+09]];
    CONST robtarget Names_1640:=[[52.729,120.884,0],[0.707106781,0,0,-0.707106781],[-1,-1,0,0],[9E+09,9E+09,9E+09,9E+09,9E+09,9E+09]];
    CONST robtarget Names_1650:=[[54.769,119.337,0],[0.707106781,0,0,-0.707106781],[-1,-1,0,0],[9E+09,9E+09,9E+09,9E+09,9E+09,9E+09]];
    CONST robtarget Names_1660:=[[51.514,116.117,0],[0.707106781,0,0,-0.707106781],[-1,-1,0,0],[9E+09,9E+09,9E+09,9E+09,9E+09,9E+09]];
    CONST robtarget Names_1670:=[[48.209,115.241,0],[0.707106781,0,0,-0.707106781],[-1,-1,0,0],[9E+09,9E+09,9E+09,9E+09,9E+09,9E+09]];
    CONST robtarget Names_1680:=[[45.124,116.015,0],[0.707106781,0,0,-0.707106781],[-1,-1,0,0],[9E+09,9E+09,9E+09,9E+09,9E+09,9E+09]];
    CONST robtarget Names_1690:=[[42.923,118.131,0],[0.707106781,0,0,-0.707106781],[-1,-1,0,0],[9E+09,9E+09,9E+09,9E+09,9E+09,9E+09]];
    CONST robtarget Names_1700:=[[42.141,121.105,0],[0.707106781,0,0,-0.707106781],[-1,-1,0,0],[9E+09,9E+09,9E+09,9E+09,9E+09,9E+09]];
    CONST robtarget Names_1710:=[[43.467,124.929,0],[0.707106781,0,0,-0.707106781],[-1,-1,0,0],[9E+09,9E+09,9E+09,9E+09,9E+09,9E+09]];
    CONST robtarget Names_1720:=[[47.359,128.345,0],[0.707106781,0,0,-0.707106781],[-1,-1,0,0],[9E+09,9E+09,9E+09,9E+09,9E+09,9E+09]];
    CONST robtarget Names_1730:=[[51.642,132.356,0],[0.707106781,0,0,-0.707106781],[-1,-1,0,0],[9E+09,9E+09,9E+09,9E+09,9E+09,9E+09]];
    CONST robtarget Names_1740:=[[52.492,134.82,0],[0.707106781,0,0,-0.707106781],[-1,-1,0,0],[9E+09,9E+09,9E+09,9E+09,9E+09,9E+09]];
    CONST robtarget Names_1750:=[[51.914,136.91,0],[0.707106781,0,0,-0.707106781],[-1,-1,0,0],[9E+09,9E+09,9E+09,9E+09,9E+09,9E+09]];
    CONST robtarget Names_1760:=[[50.231,138.482,0],[0.707106781,0,0,-0.707106781],[-1,-1,0,0],[9E+09,9E+09,9E+09,9E+09,9E+09,9E+09]];
    CONST robtarget Names_1770:=[[47.869,139.069,0],[0.707106781,0,0,-0.707106781],[-1,-1,0,0],[9E+09,9E+09,9E+09,9E+09,9E+09,9E+09]];
    CONST robtarget Names_1780:=[[44.729,137.752,0],[0.707106781,0,0,-0.707106781],[-1,-1,0,0],[9E+09,9E+09,9E+09,9E+09,9E+09,9E+09]];
    CONST robtarget Names_1790:=[[42.685,134.939,0],[0.707106781,0,0,-0.707106781],[-1,-1,0,0],[9E+09,9E+09,9E+09,9E+09,9E+09,9E+09]];
    CONST robtarget Names_1800:=[[40.561,136.213,0],[0.707106781,0,0,-0.707106781],[-1,-1,0,0],[9E+09,9E+09,9E+09,9E+09,9E+09,9E+09]];
    CONST robtarget Names_1810:=[[40.561,136.213,-17],[0.707106781,0,0,-0.707106781],[-1,-1,0,0],[9E+09,9E+09,9E+09,9E+09,9E+09,9E+09]];
    CONST robtarget Names_1820:=[[68.739,141.346,-17],[0.707106781,0,0,-0.707106781],[-1,-1,0,0],[9E+09,9E+09,9E+09,9E+09,9E+09,9E+09]];
    CONST robtarget Names_1830:=[[68.739,141.346,0],[0.707106781,0,0,-0.707106781],[-1,-1,0,0],[9E+09,9E+09,9E+09,9E+09,9E+09,9E+09]];
    CONST robtarget Names_1840:=[[65.087,140.629,0],[0.707106781,0,0,-0.707106781],[-1,-1,0,0],[9E+09,9E+09,9E+09,9E+09,9E+09,9E+09]];
    CONST robtarget Names_1850:=[[62.034,138.499,0],[0.707106781,0,0,-0.707106781],[-1,-1,0,0],[9E+09,9E+09,9E+09,9E+09,9E+09,9E+09]];
    CONST robtarget Names_1860:=[[59.941,135.32,0],[0.707106781,0,0,-0.707106781],[-1,-1,0,0],[9E+09,9E+09,9E+09,9E+09,9E+09,9E+09]];
    CONST robtarget Names_1870:=[[59.256,131.574,0],[0.707106781,0,0,-0.707106781],[-1,-1,0,0],[9E+09,9E+09,9E+09,9E+09,9E+09,9E+09]];
    CONST robtarget Names_1880:=[[59.956,127.87,0],[0.707106781,0,0,-0.707106781],[-1,-1,0,0],[9E+09,9E+09,9E+09,9E+09,9E+09,9E+09]];
    CONST robtarget Names_1890:=[[62.06,124.742,0],[0.707106781,0,0,-0.707106781],[-1,-1,0,0],[9E+09,9E+09,9E+09,9E+09,9E+09,9E+09]];
    CONST robtarget Names_1900:=[[65.137,122.618,0],[0.707106781,0,0,-0.707106781],[-1,-1,0,0],[9E+09,9E+09,9E+09,9E+09,9E+09,9E+09]];
    CONST robtarget Names_1910:=[[68.807,121.903,0],[0.707106781,0,0,-0.707106781],[-1,-1,0,0],[9E+09,9E+09,9E+09,9E+09,9E+09,9E+09]];
    CONST robtarget Names_1920:=[[72.928,122.872,0],[0.707106781,0,0,-0.707106781],[-1,-1,0,0],[9E+09,9E+09,9E+09,9E+09,9E+09,9E+09]];
    CONST robtarget Names_1930:=[[76.166,125.778,0],[0.707106781,0,0,-0.707106781],[-1,-1,0,0],[9E+09,9E+09,9E+09,9E+09,9E+09,9E+09]];
    CONST robtarget Names_1940:=[[76.166,122.379,0],[0.707106781,0,0,-0.707106781],[-1,-1,0,0],[9E+09,9E+09,9E+09,9E+09,9E+09,9E+09]];
    CONST robtarget Names_1950:=[[78.511,122.379,0],[0.707106781,0,0,-0.707106781],[-1,-1,0,0],[9E+09,9E+09,9E+09,9E+09,9E+09,9E+09]];
    CONST robtarget Names_1960:=[[78.511,140.87,0],[0.707106781,0,0,-0.707106781],[-1,-1,0,0],[9E+09,9E+09,9E+09,9E+09,9E+09,9E+09]];
    CONST robtarget Names_1970:=[[76.166,140.87,0],[0.707106781,0,0,-0.707106781],[-1,-1,0,0],[9E+09,9E+09,9E+09,9E+09,9E+09,9E+09]];
    CONST robtarget Names_1980:=[[76.166,137.692,0],[0.707106781,0,0,-0.707106781],[-1,-1,0,0],[9E+09,9E+09,9E+09,9E+09,9E+09,9E+09]];
    CONST robtarget Names_1990:=[[72.809,140.428,0],[0.707106781,0,0,-0.707106781],[-1,-1,0,0],[9E+09,9E+09,9E+09,9E+09,9E+09,9E+09]];
    CONST robtarget Names_2000:=[[68.739,141.346,0],[0.707106781,0,0,-0.707106781],[-1,-1,0,0],[9E+09,9E+09,9E+09,9E+09,9E+09,9E+09]];
    CONST robtarget Names_2010:=[[68.739,141.346,-17],[0.707106781,0,0,-0.707106781],[-1,-1,0,0],[9E+09,9E+09,9E+09,9E+09,9E+09,9E+09]];
    CONST robtarget Names_2020:=[[83.865,140.87,-17],[0.608761429,0,0,-0.79335334],[-1,0,-1,0],[9E+09,9E+09,9E+09,9E+09,9E+09,9E+09]];
    CONST robtarget Names_2030:=[[83.865,140.87,0],[0.608761429,0,0,-0.79335334],[-1,0,-1,0],[9E+09,9E+09,9E+09,9E+09,9E+09,9E+09]];
    CONST robtarget Names_2040:=[[83.865,122.379,0],[0.608761429,0,0,-0.79335334],[-1,0,-1,0],[9E+09,9E+09,9E+09,9E+09,9E+09,9E+09]];
    CONST robtarget Names_2050:=[[86.244,122.379,0],[0.608761429,0,0,-0.79335334],[-1,0,-1,0],[9E+09,9E+09,9E+09,9E+09,9E+09,9E+09]];
    CONST robtarget Names_2060:=[[86.244,125.693,0],[0.608761429,0,0,-0.79335334],[-1,0,-1,0],[9E+09,9E+09,9E+09,9E+09,9E+09,9E+09]];
    CONST robtarget Names_2070:=[[89.405,122.847,0],[0.608761429,0,0,-0.79335334],[-1,0,-1,0],[9E+09,9E+09,9E+09,9E+09,9E+09,9E+09]];
    CONST robtarget Names_2080:=[[93.178,121.903,0],[0.608761429,0,0,-0.79335334],[-1,0,-1,0],[9E+09,9E+09,9E+09,9E+09,9E+09,9E+09]];
    CONST robtarget Names_2090:=[[96.858,122.957,0],[0.608761429,0,0,-0.79335334],[-1,0,-1,0],[9E+09,9E+09,9E+09,9E+09,9E+09,9E+09]];
    CONST robtarget Names_2100:=[[99.228,125.795,0],[0.608761429,0,0,-0.79335334],[-1,0,-1,0],[9E+09,9E+09,9E+09,9E+09,9E+09,9E+09]];
    CONST robtarget Names_2110:=[[99.993,131.353,0],[0.608761429,0,0,-0.79335334],[-1,0,-1,0],[9E+09,9E+09,9E+09,9E+09,9E+09,9E+09]];
    CONST robtarget Names_2120:=[[99.993,140.87,0],[0.608761429,0,0,-0.79335334],[-1,0,-1,0],[9E+09,9E+09,9E+09,9E+09,9E+09,9E+09]];
    CONST robtarget Names_2130:=[[97.614,140.87,0],[0.608761429,0,0,-0.79335334],[-1,0,-1,0],[9E+09,9E+09,9E+09,9E+09,9E+09,9E+09]];
    CONST robtarget Names_2140:=[[97.614,132.05,0],[0.608761429,0,0,-0.79335334],[-1,0,-1,0],[9E+09,9E+09,9E+09,9E+09,9E+09,9E+09]];
    CONST robtarget Names_2150:=[[97.349,127.784,0],[0.608761429,0,0,-0.79335334],[-1,0,-1,0],[9E+09,9E+09,9E+09,9E+09,9E+09,9E+09]];
    CONST robtarget Names_2160:=[[95.763,125.022,0],[0.608761429,0,0,-0.79335334],[-1,0,-1,0],[9E+09,9E+09,9E+09,9E+09,9E+09,9E+09]];
    CONST robtarget Names_2170:=[[92.703,124.096,0],[0.608761429,0,0,-0.79335334],[-1,0,-1,0],[9E+09,9E+09,9E+09,9E+09,9E+09,9E+09]];
    CONST robtarget Names_2180:=[[88.836,125.523,0],[0.608761429,0,0,-0.79335334],[-1,0,-1,0],[9E+09,9E+09,9E+09,9E+09,9E+09,9E+09]];
    CONST robtarget Names_2190:=[[86.584,129.058,0],[0.608761429,0,0,-0.79335334],[-1,0,-1,0],[9E+09,9E+09,9E+09,9E+09,9E+09,9E+09]];
    CONST robtarget Names_2200:=[[86.244,134.089,0],[0.608761429,0,0,-0.79335334],[-1,0,-1,0],[9E+09,9E+09,9E+09,9E+09,9E+09,9E+09]];
    CONST robtarget Names_2210:=[[86.244,140.87,0],[0.608761429,0,0,-0.79335334],[-1,0,-1,0],[9E+09,9E+09,9E+09,9E+09,9E+09,9E+09]];
    CONST robtarget Names_2220:=[[83.865,140.87,0],[0.608761429,0,0,-0.79335334],[-1,0,-1,0],[9E+09,9E+09,9E+09,9E+09,9E+09,9E+09]];
    CONST robtarget Names_2230:=[[83.865,140.87,-17],[0.608761429,0,0,-0.79335334],[-1,0,-1,0],[9E+09,9E+09,9E+09,9E+09,9E+09,9E+09]];
    CONST robtarget Names_2250:=[[107.165,140.87,-17],[0.608761429,0,0,-0.79335334],[-1,0,-1,0],[9E+09,9E+09,9E+09,9E+09,9E+09,9E+09]];
    CONST robtarget Names_2260:=[[107.165,140.87,0],[0.608761429,0,0,-0.79335334],[-1,0,-1,0],[9E+09,9E+09,9E+09,9E+09,9E+09,9E+09]];
    CONST robtarget Names_2270:=[[107.165,124.436,0],[0.608761429,0,0,-0.79335334],[-1,0,-1,0],[9E+09,9E+09,9E+09,9E+09,9E+09,9E+09]];
    CONST robtarget Names_2280:=[[103.919,124.436,0],[0.608761429,0,0,-0.79335334],[-1,0,-1,0],[9E+09,9E+09,9E+09,9E+09,9E+09,9E+09]];
    CONST robtarget Names_2290:=[[103.919,122.379,0],[0.608761429,0,0,-0.79335334],[-1,0,-1,0],[9E+09,9E+09,9E+09,9E+09,9E+09,9E+09]];
    CONST robtarget Names_2300:=[[107.165,122.379,0],[0.608761429,0,0,-0.79335334],[-1,0,-1,0],[9E+09,9E+09,9E+09,9E+09,9E+09,9E+09]];
    CONST robtarget Names_2310:=[[107.165,115.513,0],[0.608761429,0,0,-0.79335334],[-1,0,-1,0],[9E+09,9E+09,9E+09,9E+09,9E+09,9E+09]];
    CONST robtarget Names_2320:=[[109.545,115.513,0],[0.608761429,0,0,-0.79335334],[-1,0,-1,0],[9E+09,9E+09,9E+09,9E+09,9E+09,9E+09]];
    CONST robtarget Names_2330:=[[109.545,122.379,0],[0.608761429,0,0,-0.79335334],[-1,0,-1,0],[9E+09,9E+09,9E+09,9E+09,9E+09,9E+09]];
    CONST robtarget Names_2340:=[[113.317,122.379,0],[0.608761429,0,0,-0.79335334],[-1,0,-1,0],[9E+09,9E+09,9E+09,9E+09,9E+09,9E+09]];
    CONST robtarget Names_2350:=[[113.317,124.436,0],[0.608761429,0,0,-0.79335334],[-1,0,-1,0],[9E+09,9E+09,9E+09,9E+09,9E+09,9E+09]];
    CONST robtarget Names_2360:=[[109.545,124.436,0],[0.608761429,0,0,-0.79335334],[-1,0,-1,0],[9E+09,9E+09,9E+09,9E+09,9E+09,9E+09]];
    CONST robtarget Names_2370:=[[109.545,140.87,0],[0.608761429,0,0,-0.79335334],[-1,0,-1,0],[9E+09,9E+09,9E+09,9E+09,9E+09,9E+09]];
    CONST robtarget Names_2380:=[[107.165,140.87,0],[0.608761429,0,0,-0.79335334],[-1,0,-1,0],[9E+09,9E+09,9E+09,9E+09,9E+09,9E+09]];
    CONST robtarget Names_2390:=[[107.165,140.87,-17],[0.608761429,0,0,-0.79335334],[-1,0,-1,0],[9E+09,9E+09,9E+09,9E+09,9E+09,9E+09]];
    CONST robtarget Names_2400:=[[117.711,118.691,-17],[0.608761429,0,0,-0.79335334],[-1,0,-1,0],[9E+09,9E+09,9E+09,9E+09,9E+09,9E+09]];
    CONST robtarget Names_2410:=[[117.711,118.691,0],[0.608761429,0,0,-0.79335334],[-1,0,-1,0],[9E+09,9E+09,9E+09,9E+09,9E+09,9E+09]];
    CONST robtarget Names_2420:=[[116.34,118.114,0],[0.608761429,0,0,-0.79335334],[-1,0,-1,0],[9E+09,9E+09,9E+09,9E+09,9E+09,9E+09]];
    CONST robtarget Names_2430:=[[115.765,116.737,0],[0.608761429,0,0,-0.79335334],[-1,0,-1,0],[9E+09,9E+09,9E+09,9E+09,9E+09,9E+09]];
    CONST robtarget Names_2440:=[[116.34,115.343,0],[0.608761429,0,0,-0.79335334],[-1,0,-1,0],[9E+09,9E+09,9E+09,9E+09,9E+09,9E+09]];
    CONST robtarget Names_2450:=[[117.711,114.765,0],[0.608761429,0,0,-0.79335334],[-1,0,-1,0],[9E+09,9E+09,9E+09,9E+09,9E+09,9E+09]];
    CONST robtarget Names_2460:=[[119.098,115.343,0],[0.608761429,0,0,-0.79335334],[-1,0,-1,0],[9E+09,9E+09,9E+09,9E+09,9E+09,9E+09]];
    CONST robtarget Names_2470:=[[119.674,116.737,0],[0.608761429,0,0,-0.79335334],[-1,0,-1,0],[9E+09,9E+09,9E+09,9E+09,9E+09,9E+09]];
    CONST robtarget Names_2480:=[[119.098,118.114,0],[0.608761429,0,0,-0.79335334],[-1,0,-1,0],[9E+09,9E+09,9E+09,9E+09,9E+09,9E+09]];
    CONST robtarget Names_2490:=[[117.711,118.691,0],[0.608761429,0,0,-0.79335334],[-1,0,-1,0],[9E+09,9E+09,9E+09,9E+09,9E+09,9E+09]];
    CONST robtarget Names_2500:=[[117.719,122.379,0],[0.608761429,0,0,-0.79335334],[-1,0,-1,0],[9E+09,9E+09,9E+09,9E+09,9E+09,9E+09]];
    CONST robtarget Names_2510:=[[116.53,122.379,0],[0.608761429,0,0,-0.79335334],[-1,0,-1,0],[9E+09,9E+09,9E+09,9E+09,9E+09,9E+09]];
    CONST robtarget Names_2520:=[[116.53,140.87,0],[0.608761429,0,0,-0.79335334],[-1,0,-1,0],[9E+09,9E+09,9E+09,9E+09,9E+09,9E+09]];
    CONST robtarget Names_2530:=[[118.909,140.87,0],[0.608761429,0,0,-0.79335334],[-1,0,-1,0],[9E+09,9E+09,9E+09,9E+09,9E+09,9E+09]];
    CONST robtarget Names_2540:=[[118.909,122.379,0],[0.608761429,0,0,-0.79335334],[-1,0,-1,0],[9E+09,9E+09,9E+09,9E+09,9E+09,9E+09]];
    CONST robtarget Names_2550:=[[117.719,122.379,0],[0.608761429,0,0,-0.79335334],[-1,0,-1,0],[9E+09,9E+09,9E+09,9E+09,9E+09,9E+09]];
    CONST robtarget Names_2560:=[[117.719,122.379,-17],[0.608761429,0,0,-0.79335334],[-1,0,-1,0],[9E+09,9E+09,9E+09,9E+09,9E+09,9E+09]];
    CONST robtarget Names_2570:=[[132.505,141.346,-17],[0.608761429,0,0,-0.79335334],[-1,0,-1,0],[9E+09,9E+09,9E+09,9E+09,9E+09,9E+09]];
    CONST robtarget Names_2580:=[[132.505,141.346,0],[0.608761429,0,0,-0.79335334],[-1,0,-1,0],[9E+09,9E+09,9E+09,9E+09,9E+09,9E+09]];
    CONST robtarget Names_2590:=[[128.854,140.629,0],[0.608761429,0,0,-0.79335334],[-1,0,-1,0],[9E+09,9E+09,9E+09,9E+09,9E+09,9E+09]];
    CONST robtarget Names_2600:=[[125.8,138.499,0],[0.608761429,0,0,-0.79335334],[-1,0,-1,0],[9E+09,9E+09,9E+09,9E+09,9E+09,9E+09]];
    CONST robtarget Names_2610:=[[123.707,135.32,0],[0.608761429,0,0,-0.79335334],[-1,0,-1,0],[9E+09,9E+09,9E+09,9E+09,9E+09,9E+09]];
    CONST robtarget Names_2620:=[[123.022,131.574,0],[0.608761429,0,0,-0.79335334],[-1,0,-1,0],[9E+09,9E+09,9E+09,9E+09,9E+09,9E+09]];
    CONST robtarget Names_2630:=[[123.722,127.87,0],[0.608761429,0,0,-0.79335334],[-1,0,-1,0],[9E+09,9E+09,9E+09,9E+09,9E+09,9E+09]];
    CONST robtarget Names_2640:=[[125.826,124.742,0],[0.608761429,0,0,-0.79335334],[-1,0,-1,0],[9E+09,9E+09,9E+09,9E+09,9E+09,9E+09]];
    CONST robtarget Names_2650:=[[128.904,122.618,0],[0.608761429,0,0,-0.79335334],[-1,0,-1,0],[9E+09,9E+09,9E+09,9E+09,9E+09,9E+09]];
    CONST robtarget Names_2660:=[[132.573,121.903,0],[0.608761429,0,0,-0.79335334],[-1,0,-1,0],[9E+09,9E+09,9E+09,9E+09,9E+09,9E+09]];
    CONST robtarget Names_2670:=[[136.694,122.872,0],[0.608761429,0,0,-0.79335334],[-1,0,-1,0],[9E+09,9E+09,9E+09,9E+09,9E+09,9E+09]];
    CONST robtarget Names_2680:=[[139.932,125.778,0],[0.608761429,0,0,-0.79335334],[-1,0,-1,0],[9E+09,9E+09,9E+09,9E+09,9E+09,9E+09]];
    CONST robtarget Names_2690:=[[139.932,122.379,0],[0.608761429,0,0,-0.79335334],[-1,0,-1,0],[9E+09,9E+09,9E+09,9E+09,9E+09,9E+09]];
    CONST robtarget Names_2700:=[[142.277,122.379,0],[0.608761429,0,0,-0.79335334],[-1,0,-1,0],[9E+09,9E+09,9E+09,9E+09,9E+09,9E+09]];
    CONST robtarget Names_2710:=[[142.277,140.87,0],[0.608761429,0,0,-0.79335334],[-1,0,-1,0],[9E+09,9E+09,9E+09,9E+09,9E+09,9E+09]];
    CONST robtarget Names_2720:=[[139.932,140.87,0],[0.608761429,0,0,-0.79335334],[-1,0,-1,0],[9E+09,9E+09,9E+09,9E+09,9E+09,9E+09]];
    CONST robtarget Names_2730:=[[139.932,137.692,0],[0.608761429,0,0,-0.79335334],[-1,0,-1,0],[9E+09,9E+09,9E+09,9E+09,9E+09,9E+09]];
    CONST robtarget Names_2740:=[[136.575,140.428,0],[0.608761429,0,0,-0.79335334],[-1,0,-1,0],[9E+09,9E+09,9E+09,9E+09,9E+09,9E+09]];
    CONST robtarget Names_2750:=[[132.505,141.346,0],[0.608761429,0,0,-0.79335334],[-1,0,-1,0],[9E+09,9E+09,9E+09,9E+09,9E+09,9E+09]];
    CONST robtarget Names_2760:=[[132.505,141.346,-17],[0.608761429,0,0,-0.79335334],[-1,0,-1,0],[9E+09,9E+09,9E+09,9E+09,9E+09,9E+09]];
    CONST robtarget Names_2770:=[[156.468,148.11,-17],[0.5,0,0,-0.866025404],[-1,0,-1,0],[9E+09,9E+09,9E+09,9E+09,9E+09,9E+09]];
    CONST robtarget Names_2780:=[[156.468,148.11,0],[0.5,0,0,-0.866025404],[-1,0,-1,0],[9E+09,9E+09,9E+09,9E+09,9E+09,9E+09]];
    CONST robtarget Names_2790:=[[152.194,147.437,0],[0.5,0,0,-0.866025404],[-1,0,-1,0],[9E+09,9E+09,9E+09,9E+09,9E+09,9E+09]];
    CONST robtarget Names_2800:=[[149.109,145.63,0],[0.5,0,0,-0.866025404],[-1,0,-1,0],[9E+09,9E+09,9E+09,9E+09,9E+09,9E+09]];
    CONST robtarget Names_2810:=[[146.917,142.315,0],[0.5,0,0,-0.866025404],[-1,0,-1,0],[9E+09,9E+09,9E+09,9E+09,9E+09,9E+09]];
    CONST robtarget Names_2820:=[[149.5,142.315,0],[0.5,0,0,-0.866025404],[-1,0,-1,0],[9E+09,9E+09,9E+09,9E+09,9E+09,9E+09]];
    CONST robtarget Names_2830:=[[152.223,145.034,0],[0.5,0,0,-0.866025404],[-1,0,-1,0],[9E+09,9E+09,9E+09,9E+09,9E+09,9E+09]];
    CONST robtarget Names_2840:=[[156.358,145.918,0],[0.5,0,0,-0.866025404],[-1,0,-1,0],[9E+09,9E+09,9E+09,9E+09,9E+09,9E+09]];
    CONST robtarget Names_2850:=[[160.467,145.012,0],[0.5,0,0,-0.866025404],[-1,0,-1,0],[9E+09,9E+09,9E+09,9E+09,9E+09,9E+09]];
    CONST robtarget Names_2860:=[[162.858,142.733,0],[0.5,0,0,-0.866025404],[-1,0,-1,0],[9E+09,9E+09,9E+09,9E+09,9E+09,9E+09]];
    CONST robtarget Names_2870:=[[163.572,138.304,0],[0.5,0,0,-0.866025404],[-1,0,-1,0],[9E+09,9E+09,9E+09,9E+09,9E+09,9E+09]];
    CONST robtarget Names_2880:=[[163.572,137.352,0],[0.5,0,0,-0.866025404],[-1,0,-1,0],[9E+09,9E+09,9E+09,9E+09,9E+09,9E+09]];
    CONST robtarget Names_2890:=[[160.289,139.961,0],[0.5,0,0,-0.866025404],[-1,0,-1,0],[9E+09,9E+09,9E+09,9E+09,9E+09,9E+09]];
    CONST robtarget Names_2900:=[[156.172,140.87,0],[0.5,0,0,-0.866025404],[-1,0,-1,0],[9E+09,9E+09,9E+09,9E+09,9E+09,9E+09]];
    CONST robtarget Names_2910:=[[151.374,139.604,0],[0.5,0,0,-0.866025404],[-1,0,-1,0],[9E+09,9E+09,9E+09,9E+09,9E+09,9E+09]];
    CONST robtarget Names_2920:=[[147.904,136.196,0],[0.5,0,0,-0.866025404],[-1,0,-1,0],[9E+09,9E+09,9E+09,9E+09,9E+09,9E+09]];
    CONST robtarget Names_2930:=[[146.679,131.489,0],[0.5,0,0,-0.866025404],[-1,0,-1,0],[9E+09,9E+09,9E+09,9E+09,9E+09,9E+09]];
    CONST robtarget Names_2940:=[[147.955,126.705,0],[0.5,0,0,-0.866025404],[-1,0,-1,0],[9E+09,9E+09,9E+09,9E+09,9E+09,9E+09]];
    CONST robtarget Names_2950:=[[151.485,123.195,0],[0.5,0,0,-0.866025404],[-1,0,-1,0],[9E+09,9E+09,9E+09,9E+09,9E+09,9E+09]];
    CONST robtarget Names_2960:=[[156.24,121.903,0],[0.5,0,0,-0.866025404],[-1,0,-1,0],[9E+09,9E+09,9E+09,9E+09,9E+09,9E+09]];
    CONST robtarget Names_2970:=[[160.11,122.762,0],[0.5,0,0,-0.866025404],[-1,0,-1,0],[9E+09,9E+09,9E+09,9E+09,9E+09,9E+09]];
    CONST robtarget Names_2980:=[[163.572,125.591,0],[0.5,0,0,-0.866025404],[-1,0,-1,0],[9E+09,9E+09,9E+09,9E+09,9E+09,9E+09]];
    CONST robtarget Names_2990:=[[163.572,122.379,0],[0.5,0,0,-0.866025404],[-1,0,-1,0],[9E+09,9E+09,9E+09,9E+09,9E+09,9E+09]];
    CONST robtarget Names_3000:=[[165.952,122.379,0],[0.5,0,0,-0.866025404],[-1,0,-1,0],[9E+09,9E+09,9E+09,9E+09,9E+09,9E+09]];
    CONST robtarget Names_3010:=[[165.952,137.114,0],[0.5,0,0,-0.866025404],[-1,0,-1,0],[9E+09,9E+09,9E+09,9E+09,9E+09,9E+09]];
    CONST robtarget Names_3020:=[[165.272,142.808,0],[0.5,0,0,-0.866025404],[-1,0,-1,0],[9E+09,9E+09,9E+09,9E+09,9E+09,9E+09]];
    CONST robtarget Names_3030:=[[162.026,146.734,0],[0.5,0,0,-0.866025404],[-1,0,-1,0],[9E+09,9E+09,9E+09,9E+09,9E+09,9E+09]];
    CONST robtarget Names_3040:=[[156.468,148.11,0],[0.5,0,0,-0.866025404],[-1,0,-1,0],[9E+09,9E+09,9E+09,9E+09,9E+09,9E+09]];
    CONST robtarget Names_3050:=[[156.468,148.11,-17],[0.5,0,0,-0.866025404],[-1,0,-1,0],[9E+09,9E+09,9E+09,9E+09,9E+09,9E+09]];
    CONST robtarget Names_3060:=[[179.803,141.346,-17],[0.5,0,0,-0.866025404],[-1,0,-1,0],[9E+09,9E+09,9E+09,9E+09,9E+09,9E+09]];
    CONST robtarget Names_3070:=[[179.803,141.346,0],[0.5,0,0,-0.866025404],[-1,0,-1,0],[9E+09,9E+09,9E+09,9E+09,9E+09,9E+09]];
    CONST robtarget Names_3080:=[[176.007,140.651,0],[0.5,0,0,-0.866025404],[-1,0,-1,0],[9E+09,9E+09,9E+09,9E+09,9E+09,9E+09]];
    CONST robtarget Names_3090:=[[172.848,138.448,0],[0.5,0,0,-0.866025404],[-1,0,-1,0],[9E+09,9E+09,9E+09,9E+09,9E+09,9E+09]];
    CONST robtarget Names_3100:=[[170.832,135.327,0],[0.5,0,0,-0.866025404],[-1,0,-1,0],[9E+09,9E+09,9E+09,9E+09,9E+09,9E+09]];
    CONST robtarget Names_3110:=[[170.15,131.676,0],[0.5,0,0,-0.866025404],[-1,0,-1,0],[9E+09,9E+09,9E+09,9E+09,9E+09,9E+09]];
    CONST robtarget Names_3120:=[[170.785,128.098,0],[0.5,0,0,-0.866025404],[-1,0,-1,0],[9E+09,9E+09,9E+09,9E+09,9E+09,9E+09]];
    CONST robtarget Names_3130:=[[172.703,125.014,0],[0.5,0,0,-0.866025404],[-1,0,-1,0],[9E+09,9E+09,9E+09,9E+09,9E+09,9E+09]];
    CONST robtarget Names_3140:=[[175.907,122.671,0],[0.5,0,0,-0.866025404],[-1,0,-1,0],[9E+09,9E+09,9E+09,9E+09,9E+09,9E+09]];
    CONST robtarget Names_3150:=[[179.803,121.903,0],[0.5,0,0,-0.866025404],[-1,0,-1,0],[9E+09,9E+09,9E+09,9E+09,9E+09,9E+09]];
    CONST robtarget Names_3160:=[[183.687,122.667,0],[0.5,0,0,-0.866025404],[-1,0,-1,0],[9E+09,9E+09,9E+09,9E+09,9E+09,9E+09]];
    CONST robtarget Names_3170:=[[186.885,124.997,0],[0.5,0,0,-0.866025404],[-1,0,-1,0],[9E+09,9E+09,9E+09,9E+09,9E+09,9E+09]];
    CONST robtarget Names_3180:=[[188.806,128.09,0],[0.5,0,0,-0.866025404],[-1,0,-1,0],[9E+09,9E+09,9E+09,9E+09,9E+09,9E+09]];
    CONST robtarget Names_3190:=[[189.439,131.676,0],[0.5,0,0,-0.866025404],[-1,0,-1,0],[9E+09,9E+09,9E+09,9E+09,9E+09,9E+09]];
    CONST robtarget Names_3200:=[[188.756,135.327,0],[0.5,0,0,-0.866025404],[-1,0,-1,0],[9E+09,9E+09,9E+09,9E+09,9E+09,9E+09]];
    CONST robtarget Names_3210:=[[186.741,138.448,0],[0.5,0,0,-0.866025404],[-1,0,-1,0],[9E+09,9E+09,9E+09,9E+09,9E+09,9E+09]];
    CONST robtarget Names_3220:=[[183.59,140.65,0],[0.5,0,0,-0.866025404],[-1,0,-1,0],[9E+09,9E+09,9E+09,9E+09,9E+09,9E+09]];
    CONST robtarget Names_3230:=[[179.803,141.346,0],[0.5,0,0,-0.866025404],[-1,0,-1,0],[9E+09,9E+09,9E+09,9E+09,9E+09,9E+09]];
    CONST robtarget Names_3240:=[[179.803,141.346,-17],[0.5,0,0,-0.866025404],[-1,0,-1,0],[9E+09,9E+09,9E+09,9E+09,9E+09,9E+09]];

    CONST robtarget T_Maintenance:=[[-35.000037155,-1480.000027214,141.00001121],[0.707106797,-0.000000016,-0.000000016,0.707106766],[1,-1,0,0],[9E+09,9E+09,9E+09,9E+09,9E+09,9E+09]];
    !Tool
    PERS tooldata Marker:=[TRUE,[[50.065,0,105.484],[0.866025404,0,0.5,0]],[0.1,[0,0,1],[1,0,0,0],0,0,0]];
    !WorkObjects
    TASK PERS wobjdata Cake:=[FALSE,TRUE,"",[[250,0,0],[1,0,0,0]],[[-315,-605,568],[0,1,0,0]]];
    TASK PERS wobjdata Cake2:=[FALSE,TRUE,"",[[-250,0,0],[1,0,0,0]],[[-65,-605,568],[0,1,0,0]]];
    PERS wobjdata Current_Wobj:=[FALSE,TRUE,"",[[250,0,0],[1,0,0,0]],[[-315,-605,568],[0,1,0,0]]];  ! Variable de trabajo

    PROC main()
        !Var init
        SetDO DO_01, 0;
        !Conveyor Off
        SetDO Conveyor_INV,0;
        SetDO Conveyor_FWD,0;
        !Home Init
        Current_Wobj := Cake;  !Init Workobject, for simulation
        P_Home;
        WHILE TRUE DO
            Current_Wobj := Cake;
            IF DI_01 = 1 THEN
                !Init
                SetDO DO_01, 1;                     !Indicator: Working Routine
                P_Home;                             !Initialice interruption on home

                !Conveyor: Movement
                SetDO Conveyor_FWD, 1;              !On
                WaitTime 4.2;                       !Delay
                SetDO Conveyor_FWD,0;               !Off
                MARK;
                WaitTime 2;                         !Safe Wait Time

                !2nd Movement
                SetDO Conveyor_FWD,1;
                WaitTime 4.2;
                SetDO Conveyor_FWD,0;
                !Rutine End

                WaitTime 2;
                SetDO DO_01,0;                        !Indicator off: End Routine

                !Backwards Movement
                SetDO Conveyor_INV,1;
                WaitTime 8.5;
                SetDO Conveyor_INV,0;

                !Just for Simulation
                Current_Wobj := Cake2;
                WaitTime 1;
                MARK;
                WaitTime 1;

            ELSEIF DI_02 = 1 THEN
                SetDO DO_02, 1;
                P_Home;
                WaitTime 1;
                SetDO DO_02, 0;
            ELSEIF DI_03 = 1 THEN
                SetDO DO_03, 1;
                P_Maintenance;
                WaitTime 1;
                SetDO DO_03, 0;
             ENDIF
        ENDWHILE
    ENDPROC

    !SubRoutine: Paths
    PROC MARK()
        P_Home;
        !Drawing
        P_Local_Home;
        P_Bat;
        P_Local_Home;   !Local Home: Target ref to Current_Wobj (Workobj.) Bat Icon Draw
        P_Names;
        P_Local_Home;
        P_Home;       !Names Draw -> Local -> Home
    ENDPROC
    PROC P_Home()
        MoveJ T_Home,v200,z1,Marker\WObj:=Current_Wobj;
    ENDPROC
    PROC P_Bat()
        MoveL [[44.887375283,23.575,0],[0.707106781,0,0,-0.707106781],[0,0,0,0],[9E+09,9E+09,9E+09,9E+09,9E+09,9E+09]],v50,z1,Marker\WObj:=Current_Wobj;
        MoveL [[92.217626762,23.834877014,0],[0.5,0,0,-0.866025404],[-1,0,-1,0],[9E+09,9E+09,9E+09,9E+09,9E+09,9E+09]],v50,z1,Marker\WObj:=Current_Wobj;
        MoveC [[97.860623741,32.777873993,0],[0.5,0,0,-0.866025404],[-1,0,-1,0],[9E+09,9E+09,9E+09,9E+09,9E+09,9E+09]],[[109.794252014,32.852127266,0],[0.5,0,0,-0.866025404],[0,0,0,0],[9E+09,9E+09,9E+09,9E+09,9E+09,9E+09]],v50,z1,Marker\WObj:=Current_Wobj;
        MoveL [[111.283377266,25.744747734,0],[0.5,0,0,-0.866025404],[-1,0,-1,0],[9E+09,9E+09,9E+09,9E+09,9E+09,9E+09]],v50,z1,Marker\WObj:=Current_Wobj;
        MoveC [[112.525,30.426625252,0],[0.5,0,0,-0.866025404],[-1,0,-1,0],[9E+09,9E+09,9E+09,9E+09,9E+09,9E+09]],[[118.898123741,25.740625,0],[0.5,0,0,-0.866025404],[0,0,0,0],[9E+09,9E+09,9E+09,9E+09,9E+09,9E+09]],v50,z1,Marker\WObj:=Current_Wobj;
        MoveL [[120.205747986,32.852127266,0],[0.5,0,0,-0.866025404],[-1,0,-1,0],[9E+09,9E+09,9E+09,9E+09,9E+09,9E+09]],v50,z1,Marker\WObj:=Current_Wobj;
        MoveC [[132.139376259,32.777873993,0],[0.5,0,0,-0.866025404],[-1,0,-1,0],[9E+09,9E+09,9E+09,9E+09,9E+09,9E+09]],[[138.079373741,23.575,0],[0.5,0,0,-0.866025404],[0,0,0,0],[9E+09,9E+09,9E+09,9E+09,9E+09,9E+09]],v50,z1,Marker\WObj:=Current_Wobj;
        MoveL [[185.145619965,23.789501762,0],[0.5,0,0,-0.866025404],[-1,0,-1,0],[9E+09,9E+09,9E+09,9E+09,9E+09,9E+09]],v50,z1,Marker\WObj:=Current_Wobj;
        MoveC [[168.340891695,33.478608179,0],[0.5,0,0,-0.866025404],[-1,0,-1,0],[9E+09,9E+09,9E+09,9E+09,9E+09,9E+09]],[[163.773995972,51.414627266,0],[0.5,0,0,-0.866025404],[0,0,0,0],[9E+09,9E+09,9E+09,9E+09,9E+09,9E+09]],v50,z1,Marker\WObj:=Current_Wobj;
        MoveC [[135.262514114,52.897562122,0],[0.5,0,0,-0.866025404],[-1,0,-1,0],[9E+09,9E+09,9E+09,9E+09,9E+09,9E+09]],[[118.021503486,64.425747652,0],[0.5,0,0,-0.866025404],[0,0,0,0],[9E+09,9E+09,9E+09,9E+09,9E+09,9E+09]],v50,z1,Marker\WObj:=Current_Wobj;
        MoveL [[114.884500504,71.210504532,0],[0.5,0,0,-0.866025404],[-1,0,-1,0],[9E+09,9E+09,9E+09,9E+09,9E+09,9E+09]],v50,z1,Marker\WObj:=Current_Wobj;
        MoveC [[101.522546531,55.448907324,0],[0.5,0,0,-0.866025404],[-1,0,-1,0],[9E+09,9E+09,9E+09,9E+09,9E+09,9E+09]],[[79.985840188,50.770867258,0],[0.5,0,0,-0.866025404],[0,0,0,0],[9E+09,9E+09,9E+09,9E+09,9E+09,9E+09]],v50,z1,Marker\WObj:=Current_Wobj;
        MoveL [[66.061000252,51.208377266,0],[0.5,0,0,-0.866025404],[-1,0,-1,0],[9E+09,9E+09,9E+09,9E+09,9E+09,9E+09]],v50,z1,Marker\WObj:=Current_Wobj;
        MoveC [[61.659109682,33.478608179,0],[0.5,0,0,-0.866025404],[-1,0,-1,0],[9E+09,9E+09,9E+09,9E+09,9E+09,9E+09]],[[44.854375315,23.789501762,0],[0.707106781,0,0,-0.707106781],[0,0,0,0],[9E+09,9E+09,9E+09,9E+09,9E+09,9E+09]],v50,z1,Marker\WObj:=Current_Wobj;
    ENDPROC
    PROC P_Local_Home()
        MoveL T_Local_Home,v100,z1,Marker\WObj:=Current_Wobj;
    ENDPROC
    PROC P_Names()
        MoveL Names_00,v50,z1,Marker\WObj:=Current_Wobj;
        MoveL Names_10,v50,z1,Marker\WObj:=Current_Wobj;
        MoveL Names_20,v50,z1,Marker\WObj:=Current_Wobj;
        MoveC Names_30,Names_40,v50,z1,Marker\WObj:=Current_Wobj;
        MoveC Names_50,Names_60,v50,z1,Marker\WObj:=Current_Wobj;
        MoveC Names_70,Names_80,v50,z1,Marker\WObj:=Current_Wobj;
        MoveC Names_90,Names_100,v50,z1,Marker\WObj:=Current_Wobj;
        MoveC Names_110,Names_120,v50,z1,Marker\WObj:=Current_Wobj;
        MoveC Names_130,Names_140,v50,z1,Marker\WObj:=Current_Wobj;
        MoveL Names_150,v50,z1,Marker\WObj:=Current_Wobj;
        MoveL Names_160,v50,z1,Marker\WObj:=Current_Wobj;
        MoveC Names_170,Names_180,v50,z1,Marker\WObj:=Current_Wobj;
        MoveC Names_190,Names_200,v50,z1,Marker\WObj:=Current_Wobj;
        MoveC Names_210,Names_220,v50,z1,Marker\WObj:=Current_Wobj;
        MoveL Names_230,v50,z1,Marker\WObj:=Current_Wobj;
        MoveC Names_240,Names_250,v50,z1,Marker\WObj:=Current_Wobj;
        MoveC Names_260,Names_270,v50,z1,Marker\WObj:=Current_Wobj;
        MoveC Names_280,Names_290,v50,z1,Marker\WObj:=Current_Wobj;
        MoveL Names_300,v50,z1,Marker\WObj:=Current_Wobj;
        MoveL Names_310,v50,z1,Marker\WObj:=Current_Wobj;
        MoveL Names_320,v50,z1,Marker\WObj:=Current_Wobj;
        MoveL Names_330,v50,z1,Marker\WObj:=Current_Wobj;
        MoveL Names_340,v50,z1,Marker\WObj:=Current_Wobj;
        MoveC Names_350,Names_360,v50,z1,Marker\WObj:=Current_Wobj;
        MoveC Names_370,Names_380,v50,z1,Marker\WObj:=Current_Wobj;
        MoveC Names_390,Names_400,v50,z1,Marker\WObj:=Current_Wobj;
        MoveC Names_410,Names_420,v50,z1,Marker\WObj:=Current_Wobj;
        MoveC Names_430,Names_440,v50,z1,Marker\WObj:=Current_Wobj;
        MoveL Names_450,v50,z1,Marker\WObj:=Current_Wobj;
        MoveL Names_460,v50,z1,Marker\WObj:=Current_Wobj;
        MoveL Names_470,v50,z1,Marker\WObj:=Current_Wobj;
        MoveL Names_480,v50,z1,Marker\WObj:=Current_Wobj;
        MoveL Names_490,v50,z1,Marker\WObj:=Current_Wobj;
        MoveL Names_500,v50,z1,Marker\WObj:=Current_Wobj;
        MoveL Names_510,v50,z1,Marker\WObj:=Current_Wobj;
        MoveL Names_520,v50,z1,Marker\WObj:=Current_Wobj;
        MoveL Names_530,v50,z1,Marker\WObj:=Current_Wobj;
        MoveL Names_540,v50,z1,Marker\WObj:=Current_Wobj;
        MoveL Names_550,v50,z1,Marker\WObj:=Current_Wobj;
        MoveL Names_560,v50,z1,Marker\WObj:=Current_Wobj;
        MoveC Names_570,Names_580,v50,z1,Marker\WObj:=Current_Wobj;
        MoveC Names_590,Names_600,v50,z1,Marker\WObj:=Current_Wobj;
        MoveL Names_610,v50,z1,Marker\WObj:=Current_Wobj;
        MoveC Names_620,Names_630,v50,z1,Marker\WObj:=Current_Wobj;
        MoveC Names_640,Names_650,v50,z1,Marker\WObj:=Current_Wobj;
        MoveL Names_660,v50,z1,Marker\WObj:=Current_Wobj;
        MoveL Names_670,v50,z1,Marker\WObj:=Current_Wobj;
        MoveL Names_680,v50,z1,Marker\WObj:=Current_Wobj;
        MoveC Names_690,Names_700,v50,z1,Marker\WObj:=Current_Wobj;
        MoveC Names_710,Names_720,v50,z1,Marker\WObj:=Current_Wobj;
        MoveC Names_730,Names_740,v50,z1,Marker\WObj:=Current_Wobj;
        MoveC Names_750,Names_760,v50,z1,Marker\WObj:=Current_Wobj;
        MoveL Names_770,v50,z1,Marker\WObj:=Current_Wobj;
        MoveC Names_780,Names_790,v50,z1,Marker\WObj:=Current_Wobj;
        MoveC Names_800,Names_810,v50,z1,Marker\WObj:=Current_Wobj;
        MoveC Names_820,Names_830,v50,z1,Marker\WObj:=Current_Wobj;
        MoveL Names_840,v50,z1,Marker\WObj:=Current_Wobj;
        MoveL Names_850,v50,z1,Marker\WObj:=Current_Wobj;
        MoveL Names_860,v50,z1,Marker\WObj:=Current_Wobj;
        MoveL Names_870,v50,z1,Marker\WObj:=Current_Wobj;
        MoveL Names_880,v50,z1,Marker\WObj:=Current_Wobj;
        MoveL Names_890,v50,z1,Marker\WObj:=Current_Wobj;
        MoveC Names_900,Names_910,v50,z1,Marker\WObj:=Current_Wobj;
        MoveC Names_920,Names_930,v50,z1,Marker\WObj:=Current_Wobj;
        MoveL Names_940,v50,z1,Marker\WObj:=Current_Wobj;
        MoveC Names_950,Names_960,v50,z1,Marker\WObj:=Current_Wobj;
        MoveC Names_970,Names_980,v50,z1,Marker\WObj:=Current_Wobj;
        MoveC Names_990,Names_1000,v50,z1,Marker\WObj:=Current_Wobj;
        MoveC Names_1010,Names_1020,v50,z1,Marker\WObj:=Current_Wobj;
        MoveL Names_1030,v50,z1,Marker\WObj:=Current_Wobj;
        MoveC Names_1040,Names_1050,v50,z1,Marker\WObj:=Current_Wobj;
        MoveL Names_1060,v50,z1,Marker\WObj:=Current_Wobj;
        MoveL Names_1070,v50,z1,Marker\WObj:=Current_Wobj;
        MoveL Names_1080,v50,z1,Marker\WObj:=Current_Wobj;
        MoveL Names_1090,v50,z1,Marker\WObj:=Current_Wobj;
        MoveL Names_1100,v50,z1,Marker\WObj:=Current_Wobj;
        MoveL Names_1110,v50,z1,Marker\WObj:=Current_Wobj;
        MoveC Names_1120,Names_1130,v50,z1,Marker\WObj:=Current_Wobj;
        MoveC Names_1140,Names_1150,v50,z1,Marker\WObj:=Current_Wobj;
        MoveC Names_1160,Names_1170,v50,z1,Marker\WObj:=Current_Wobj;
        MoveC Names_1180,Names_1190,v50,z1,Marker\WObj:=Current_Wobj;
        MoveL Names_1200,v50,z1,Marker\WObj:=Current_Wobj;
        MoveL Names_1210,v50,z1,Marker\WObj:=Current_Wobj;
        MoveL Names_1220,v50,z1,Marker\WObj:=Current_Wobj;
        MoveC Names_1230,Names_1240,v50,z1,Marker\WObj:=Current_Wobj;
        MoveC Names_1250,Names_1260,v50,z1,Marker\WObj:=Current_Wobj;
        MoveL Names_1270,v50,z1,Marker\WObj:=Current_Wobj;
        MoveL Names_1280,v50,z1,Marker\WObj:=Current_Wobj;
        MoveL Names_1290,v50,z1,Marker\WObj:=Current_Wobj;
        MoveL Names_1300,v50,z1,Marker\WObj:=Current_Wobj;
        MoveC Names_1310,Names_1320,v50,z1,Marker\WObj:=Current_Wobj;
        MoveC Names_1330,Names_1340,v50,z1,Marker\WObj:=Current_Wobj;
        MoveC Names_1350,Names_1360,v50,z1,Marker\WObj:=Current_Wobj;
        MoveL Names_1370,v50,z1,Marker\WObj:=Current_Wobj;
        MoveL Names_1380,v50,z1,Marker\WObj:=Current_Wobj;
        MoveC Names_1390,Names_1400,v50,z1,Marker\WObj:=Current_Wobj;
        MoveL Names_1410,v50,z1,Marker\WObj:=Current_Wobj;
        MoveL Names_1420,v50,z1,Marker\WObj:=Current_Wobj;
        MoveL Names_1430,v50,z1,Marker\WObj:=Current_Wobj;
        MoveL Names_1440,v50,z1,Marker\WObj:=Current_Wobj;
        MoveL Names_1450,v50,z1,Marker\WObj:=Current_Wobj;
        MoveL Names_1460,v50,z1,Marker\WObj:=Current_Wobj;
        MoveL Names_1470,v50,z1,Marker\WObj:=Current_Wobj;
        MoveL Names_1480,v50,z1,Marker\WObj:=Current_Wobj;
        MoveL Names_1490,v50,z1,Marker\WObj:=Current_Wobj;
        MoveL Names_1500,v50,z1,Marker\WObj:=Current_Wobj;
        MoveL Names_1510,v50,z1,Marker\WObj:=Current_Wobj;
        MoveC Names_1520,Names_1530,v50,z1,Marker\WObj:=Current_Wobj;
        MoveC Names_1540,Names_1550,v50,z1,Marker\WObj:=Current_Wobj;
        MoveC Names_1560,Names_1570,v50,z1,Marker\WObj:=Current_Wobj;
        MoveC Names_1580,Names_1590,v50,z1,Marker\WObj:=Current_Wobj;
        MoveC Names_1600,Names_1610,v50,z1,Marker\WObj:=Current_Wobj;
        MoveC Names_1620,Names_1630,v50,z1,Marker\WObj:=Current_Wobj;
        MoveL Names_1640,v50,z1,Marker\WObj:=Current_Wobj;
        MoveL Names_1650,v50,z1,Marker\WObj:=Current_Wobj;
        MoveC Names_1660,Names_1670,v50,z1,Marker\WObj:=Current_Wobj;
        MoveC Names_1680,Names_1690,v50,z1,Marker\WObj:=Current_Wobj;
        MoveC Names_1700,Names_1710,v50,z1,Marker\WObj:=Current_Wobj;
        MoveL Names_1720,v50,z1,Marker\WObj:=Current_Wobj;
        MoveC Names_1730,Names_1740,v50,z1,Marker\WObj:=Current_Wobj;
        MoveC Names_1750,Names_1760,v50,z1,Marker\WObj:=Current_Wobj;
        MoveC Names_1770,Names_1780,v50,z1,Marker\WObj:=Current_Wobj;
        MoveL Names_1790,v50,z1,Marker\WObj:=Current_Wobj;
        MoveL Names_1800,v50,z1,Marker\WObj:=Current_Wobj;
        MoveL Names_1810,v50,z1,Marker\WObj:=Current_Wobj;
        MoveL Names_1820,v50,z1,Marker\WObj:=Current_Wobj;
        MoveL Names_1830,v50,z1,Marker\WObj:=Current_Wobj;
        MoveL Names_1840,v50,z1,Marker\WObj:=Current_Wobj;
        MoveC Names_1850,Names_1860,v50,z1,Marker\WObj:=Current_Wobj;
        MoveC Names_1870,Names_1880,v50,z1,Marker\WObj:=Current_Wobj;
        MoveC Names_1890,Names_1900,v50,z1,Marker\WObj:=Current_Wobj;
        MoveC Names_1910,Names_1920,v50,z1,Marker\WObj:=Current_Wobj;
        MoveL Names_1930,v50,z1,Marker\WObj:=Current_Wobj;
        MoveL Names_1940,v50,z1,Marker\WObj:=Current_Wobj;
        MoveL Names_1950,v50,z1,Marker\WObj:=Current_Wobj;
        MoveL Names_1960,v50,z1,Marker\WObj:=Current_Wobj;
        MoveL Names_1970,v50,z1,Marker\WObj:=Current_Wobj;
        MoveL Names_1980,v50,z1,Marker\WObj:=Current_Wobj;
        MoveL Names_1990,v50,z1,Marker\WObj:=Current_Wobj;
        MoveL Names_2000,v50,z1,Marker\WObj:=Current_Wobj;
        MoveL Names_2010,v50,z1,Marker\WObj:=Current_Wobj;
        MoveL Names_2020,v50,z1,Marker\WObj:=Current_Wobj;
        MoveL Names_2030,v50,z1,Marker\WObj:=Current_Wobj;
        MoveL Names_2040,v50,z1,Marker\WObj:=Current_Wobj;
        MoveL Names_2050,v50,z1,Marker\WObj:=Current_Wobj;
        MoveL Names_2060,v50,z1,Marker\WObj:=Current_Wobj;
        MoveC Names_2070,Names_2080,v50,z1,Marker\WObj:=Current_Wobj;
        MoveC Names_2090,Names_2100,v50,z1,Marker\WObj:=Current_Wobj;
        MoveL Names_2110,v50,z1,Marker\WObj:=Current_Wobj;
        MoveL Names_2120,v50,z1,Marker\WObj:=Current_Wobj;
        MoveL Names_2130,v50,z1,Marker\WObj:=Current_Wobj;
        MoveC Names_2140,Names_2150,v50,z1,Marker\WObj:=Current_Wobj;
        MoveC Names_2160,Names_2170,v50,z1,Marker\WObj:=Current_Wobj;
        MoveC Names_2180,Names_2190,v50,z1,Marker\WObj:=Current_Wobj;
        MoveL Names_2200,v50,z1,Marker\WObj:=Current_Wobj;
        MoveL Names_2210,v50,z1,Marker\WObj:=Current_Wobj;
        MoveL Names_2220,v50,z1,Marker\WObj:=Current_Wobj;
        MoveL Names_2230,v50,z1,Marker\WObj:=Current_Wobj;
        MoveL Names_2250,v50,z1,Marker\WObj:=Current_Wobj;
        MoveL Names_2260,v50,z1,Marker\WObj:=Current_Wobj;
        MoveL Names_2270,v50,z1,Marker\WObj:=Current_Wobj;
        MoveL Names_2280,v50,z1,Marker\WObj:=Current_Wobj;
        MoveL Names_2290,v50,z1,Marker\WObj:=Current_Wobj;
        MoveL Names_2300,v50,z1,Marker\WObj:=Current_Wobj;
        MoveL Names_2310,v50,z1,Marker\WObj:=Current_Wobj;
        MoveL Names_2320,v50,z1,Marker\WObj:=Current_Wobj;
        MoveL Names_2330,v50,z1,Marker\WObj:=Current_Wobj;
        MoveL Names_2340,v50,z1,Marker\WObj:=Current_Wobj;
        MoveL Names_2350,v50,z1,Marker\WObj:=Current_Wobj;
        MoveL Names_2360,v50,z1,Marker\WObj:=Current_Wobj;
        MoveL Names_2370,v50,z1,Marker\WObj:=Current_Wobj;
        MoveL Names_2380,v50,z1,Marker\WObj:=Current_Wobj;
        MoveL Names_2390,v50,z1,Marker\WObj:=Current_Wobj;
        MoveL Names_2400,v50,z1,Marker\WObj:=Current_Wobj;
        MoveL Names_2410,v50,z1,Marker\WObj:=Current_Wobj;
        MoveL Names_2420,v50,z1,Marker\WObj:=Current_Wobj;
        MoveC Names_2430,Names_2440,v50,z1,Marker\WObj:=Current_Wobj;
        MoveC Names_2450,Names_2460,v50,z1,Marker\WObj:=Current_Wobj;
        MoveC Names_2470,Names_2480,v50,z1,Marker\WObj:=Current_Wobj;
        MoveL Names_2490,v50,z1,Marker\WObj:=Current_Wobj;
        MoveL Names_2500,v50,z1,Marker\WObj:=Current_Wobj;
        MoveL Names_2510,v50,z1,Marker\WObj:=Current_Wobj;
        MoveL Names_2520,v50,z1,Marker\WObj:=Current_Wobj;
        MoveL Names_2530,v50,z1,Marker\WObj:=Current_Wobj;
        MoveL Names_2540,v50,z1,Marker\WObj:=Current_Wobj;
        MoveL Names_2550,v50,z1,Marker\WObj:=Current_Wobj;
        MoveL Names_2560,v50,z1,Marker\WObj:=Current_Wobj;
        MoveL Names_2570,v50,z1,Marker\WObj:=Current_Wobj;
        MoveL Names_2580,v50,z1,Marker\WObj:=Current_Wobj;
        MoveL Names_2590,v50,z1,Marker\WObj:=Current_Wobj;
        MoveC Names_2600,Names_2610,v50,z1,Marker\WObj:=Current_Wobj;
        MoveC Names_2620,Names_2630,v50,z1,Marker\WObj:=Current_Wobj;
        MoveC Names_2640,Names_2650,v50,z1,Marker\WObj:=Current_Wobj;
        MoveC Names_2660,Names_2670,v50,z1,Marker\WObj:=Current_Wobj;
        MoveL Names_2680,v50,z1,Marker\WObj:=Current_Wobj;
        MoveL Names_2690,v50,z1,Marker\WObj:=Current_Wobj;
        MoveL Names_2700,v50,z1,Marker\WObj:=Current_Wobj;
        MoveL Names_2710,v50,z1,Marker\WObj:=Current_Wobj;
        MoveL Names_2720,v50,z1,Marker\WObj:=Current_Wobj;
        MoveL Names_2730,v50,z1,Marker\WObj:=Current_Wobj;
        MoveL Names_2740,v50,z1,Marker\WObj:=Current_Wobj;
        MoveL Names_2750,v50,z1,Marker\WObj:=Current_Wobj;
        MoveL Names_2760,v50,z1,Marker\WObj:=Current_Wobj;
        MoveL Names_2770,v50,z1,Marker\WObj:=Current_Wobj;
        MoveL Names_2780,v50,z1,Marker\WObj:=Current_Wobj;
        MoveL Names_2790,v50,z1,Marker\WObj:=Current_Wobj;
        MoveC Names_2800,Names_2810,v50,z1,Marker\WObj:=Current_Wobj;
        MoveL Names_2820,v50,z1,Marker\WObj:=Current_Wobj;
        MoveC Names_2830,Names_2840,v50,z1,Marker\WObj:=Current_Wobj;
        MoveC Names_2850,Names_2860,v50,z1,Marker\WObj:=Current_Wobj;
        MoveL Names_2870,v50,z1,Marker\WObj:=Current_Wobj;
        MoveL Names_2880,v50,z1,Marker\WObj:=Current_Wobj;
        MoveC Names_2890,Names_2900,v50,z1,Marker\WObj:=Current_Wobj;
        MoveC Names_2910,Names_2920,v50,z1,Marker\WObj:=Current_Wobj;
        MoveL Names_2930,v50,z1,Marker\WObj:=Current_Wobj;
        MoveL Names_2940,v50,z1,Marker\WObj:=Current_Wobj;
        MoveL Names_2950,v50,z1,Marker\WObj:=Current_Wobj;
        MoveL Names_2960,v50,z1,Marker\WObj:=Current_Wobj;
        MoveL Names_2970,v50,z1,Marker\WObj:=Current_Wobj;
        MoveL Names_2980,v50,z1,Marker\WObj:=Current_Wobj;
        MoveL Names_2990,v50,z1,Marker\WObj:=Current_Wobj;
        MoveL Names_3000,v50,z1,Marker\WObj:=Current_Wobj;
        MoveC Names_3010,Names_3020,v50,z1,Marker\WObj:=Current_Wobj;
        MoveL Names_3030,v50,z1,Marker\WObj:=Current_Wobj;
        MoveL Names_3040,v50,z1,Marker\WObj:=Current_Wobj;
        MoveL Names_3050,v50,z1,Marker\WObj:=Current_Wobj;
        MoveL Names_3060,v50,z1,Marker\WObj:=Current_Wobj;
        MoveL Names_3070,v50,z1,Marker\WObj:=Current_Wobj;
        MoveL Names_3080,v50,z1,Marker\WObj:=Current_Wobj;
        MoveC Names_3090,Names_3100,v50,z1,Marker\WObj:=Current_Wobj;
        MoveC Names_3110,Names_3120,v50,z1,Marker\WObj:=Current_Wobj;
        MoveC Names_3130,Names_3140,v50,z1,Marker\WObj:=Current_Wobj;
        MoveC Names_3150,Names_3160,v50,z1,Marker\WObj:=Current_Wobj;
        MoveC Names_3170,Names_3180,v50,z1,Marker\WObj:=Current_Wobj;
        MoveC Names_3190,Names_3200,v50,z1,Marker\WObj:=Current_Wobj;
        MoveC Names_3210,Names_3220,v50,z1,Marker\WObj:=Current_Wobj;
        MoveL Names_3230,v50,z1,Marker\WObj:=Current_Wobj;
        MoveL Names_3240,v50,z1,Marker\WObj:=Current_Wobj;
    ENDPROC
    PROC P_Maintenance()
        MoveJ T_Maintenance,v300,z1,Marker\WObj:=Current_Wobj;
    ENDPROC
ENDMODULE

--- Controller Data/IRB140_6_81/RAPID/TASK1/PROGMOD/TCP_t2B7.mod ---
MODULE TCP_t2B7
	! Points are read in order of declaration.
  ! Please do not change the order of points!

  LOCAL PERS robtarget pTCP_Point1:=[[517.2705,-5.522776,300.6515],[0.499380886554718,-0.00519778858870268,0.866347849369049,0.00575591530650854],[-1,1,-2,0],[9E+09,9E+09,9E+09,9E+09,9E+09,9E+09]];
	LOCAL PERS robtarget pTCP_Point2:=[[517.4753,26.61037,296.8748],[0.494102329015732,0.329368144273758,0.796000480651855,-0.117314644157887],[0,-2,1,0],[9E+09,9E+09,9E+09,9E+09,9E+09,9E+09]];
	LOCAL PERS robtarget pTCP_Point3:=[[503.4368,-18.01744,289.8195],[0.55969101190567,-0.0462285429239273,0.825725138187408,0.0527913570404053],[-1,-3,2,0],[9E+09,9E+09,9E+09,9E+09,9E+09,9E+09]];
	LOCAL PERS robtarget pTCP_Point4:=[[507.7421,7.820115,294.2143],[0.536838114261627,0.138700500130653,0.83128809928894,-0.0390773229300976],[0,-2,1,0],[9E+09,9E+09,9E+09,9E+09,9E+09,9E+09]];

ENDMODULE

--- Controller Data/IRB140_6_81/SYSPAR/EIO.cfg ---
EIO:CFG_1.0:6:1::
#
EIO_SIGNAL:

      -Name "Conveyor_FWD" -SignalType "DO" -Label "Move" -Category "control"

      -Name "Conveyor_INV" -SignalType "DO" -Label "Back" -Category "control"

      -Name "DO_01" -SignalType "DO" -Label "Indicator_1" -Category "control"

      -Name "DI_01" -SignalType "DI" -Label "Button 1" -Category "control"

      -Name "DI_02" -SignalType "DI" -Label "Button 2" -Category "control"

      -Name "DI_03" -SignalType "DI" -Label "Button 3" -Category "control"

      -Name "DO_02" -SignalType "DO" -Label "Indicator_2" -Category "control"

      -Name "DO_03" -SignalType "DO" -Label "Indicator_3" -Category "control"
